ELSE
    // No latched run / inhibited / fault: ensure safe idle
    startSequenceRunning := FALSE;

    IF step <> 50 THEN
        lineContactor := FALSE;
    END_IF

    softstarterStart     := FALSE;
    softstarterContactor := FALSE;

    tonStartDelay(IN:=FALSE);
    tonOverlapDelay(IN:=FALSE);
    tonCurrentProof(IN:=FALSE);
    tonSSFbTimeout(IN:=FALSE);
    tonLineFbTimeout(IN:=FALSE);
    instTONSoftstartDelay(IN:=FALSE);

    IF NOT runLatch THEN
        deviceState := 'Idle (Parado)';
        step := 0;
    END_IF
END_IF


//────────────────────────────────────
// Blink generator (1 s ON / 1 s OFF)
// Gerador de pisca (1 s ligado / 1 s desligado)
//────────────────────────────────────
blinkTon(IN := TRUE, PT := T#1S);
IF blinkTon.Q THEN
    blinkTon(IN := FALSE);       // reset timer next cycle / reseta o timer no próximo ciclo
    blinkBit := NOT blinkBit;    // toggle blink bit / alterna o bit de pisca
END_IF


// =============================== Status code =======================================
// 0 = OFF
// 0-1 (alternando) = STARTING
// 1 = RUNNING
// 2 = FAULT
//==============================================================================
IF faultActive THEN
    // Fault has highest priority / Falha tem maior prioridade
    statusCode := 2;                             // FAULT

ELSIF softstarterContactor OR (softstarterContactor AND lineContactor)  THEN
    // STARTING: use blink (0/1) / PARTIDA: usa pisca (0/1)
    IF blinkBit THEN
        statusCode := 1;                         // ON (blink ON)
    ELSE
        statusCode := 0;                         // OFF (blink OFF)
    END_IF

ELSIF  lineContactor AND NOT softstarterContactor THEN
    // RUNNING: steady ON / EM FUNCIONAMENTO: ligado fixo
    statusCode := 1;                             // RUNNING

ELSE
    // OFF (stopped / idle) / Desligado (parado)
    statusCode := 0;                             // OFF
END_IF

END_FUNCTION_BLOCK

// ---- Function Blocks/PaperMachine/Auxiliary/FB_PressureControl_V1.TcPOU
(*
    FB_PressureControl_V1
    - Start pulse toggles run; Stop pulse/level forces stop
    - statusCode : INT (0=Idle, 1=Running, 2=Fault)
    - PID (OSCAT CTRL_PID) with optional reverse action
    - Input PT1 filter (OSCAT FT_PT1)
    - Engineering↔% scaling helper
    - VFD run supervision + analog feedback display (current, rpm)
    - Optional low/high pressure HOLD with hysteresis (normal-stop class)
*)

FUNCTION_BLOCK FB_PressureControl_V1
VAR_INPUT
    // ===== Sequence commands =====
    startCommand            : BOOL;            // Start pulse (toggle run)
    stopCommand             : BOOL;            // Stop pulse/level (force stop)

    // ===== Mode =====
    autoMode                : BOOL;            // TRUE=Automatic / FALSE=Manual
    reverseActing           : BOOL := FALSE;   // TRUE: increasing output decreases pressure (válvula); FALSE: direct (bomba)

    // ===== Process signals (PRESSURE) =====
    pressureFeedbackEng     : REAL;            // PV (engineering units) - Ex.: bar/kPa
    pressureSetpointEng     : REAL;            // SP (engineering units)

    // ===== Manual output (direct % to final element) =====
    manualOutputPct         : REAL;            // 0..100% manual output

    // ===== PID parameters (OSCAT CTRL_PID) =====
    kp                      : REAL := 1.0;     // proportional gain (magnitude; sign handled by reverseActing)
    tn                      : REAL := 8.0;     // integral time [s]
    tv                      : REAL := 0.0;     // derivative time [s]

    // ===== Output limits & offset =====
    outLowLimitPct          : REAL := 0.0;
    outHighLimitPct         : REAL := 100.0;
    outputOffsetPct         : REAL := 0.0;     // added to final output

    // ===== PID housekeeping =====
    resetPID                : BOOL;            // reset integrator

    // ===== Input filter (OSCAT PT1) =====
    enableInputFilter       : BOOL := TRUE;
    inputFilterTime         : TIME := T#300ms;
    inputFilterGainK        : REAL := 1.0;

    displayFilterTime       : TIME := T#20MS;	
	

    // ===== Optional scaling (engineering <-> %) =====
    enableScaling           : BOOL := TRUE;
    pLoEng                  : REAL := 0.0;     // e.g., 0 bar
    pHiEng                  : REAL := 10.0;    // e.g., 10 bar

    // ===== VFD interface & supervision =====
    vfdReady                : BOOL;            // VFD ready/healthy
    vfdRunFeedback          : BOOL;            // VFD RUN feedback
    vfdFaultFeedback        : BOOL;            // VFD fault feedback
    vfdRunFbTimeout         : TIME := T#5s;    // Timeout to receive RUN FB after start

    // ===== VFD analog feedbacks =====
    vfdCurrentFeedback      : REAL;            // Motor current [A]
    vfdEngFeedback          : REAL;            // Motor enginering feedback
    vfdTorqueFeedback       : REAL;            // Motor torque feedback
	

    // ===== SAFETY (true safety only) =====
    safetyOk                : BOOL := TRUE;    // Safety relay / chain OK
    estopOk                 : BOOL := TRUE;    // E-Stop loop OK
    guardClosedOk           : BOOL := TRUE;    // Doors/guards closed

    // ===== INTERLOCKS (process permissives) — NORMAL STOP ONLY =====
    interlock1              : BOOL := TRUE;
    interlock2              : BOOL := TRUE;
    interlock3              : BOOL := TRUE;
    interlock4              : BOOL := TRUE;
    interlock5              : BOOL := TRUE;
    interlock6              : BOOL := TRUE;

    // ===== Optional low-pressure supervision (normal-stop/hold) =====
    minPressureEnable       : BOOL := FALSE;   // Enable low-P hold
    minPressureStopEng      : REAL := 0.5;     // Trip threshold (Eng units) => stop & hold
    minPressureRestartEng   : REAL := 0.7;     // Release threshold (Eng units) => auto restart
    minPressureTripTime     : TIME := T#1s;    // P < Stop for this long to trip
    minPressureReleaseTime  : TIME := T#1s;    // P > Restart for this long to release

    // ===== Optional high-pressure supervision (normal-stop/hold) =====
    maxPressureEnable       : BOOL := FALSE;   // Enable high-P hold
    maxPressureStopEng      : REAL := 9.5;     // Trip threshold (Eng units)
    maxPressureRestartEng   : REAL := 9.2;     // Release threshold (Eng units)
    maxPressureTripTime     : TIME := T#1s;
    maxPressureReleaseTime  : TIME := T#1s;
END_VAR

VAR_OUTPUT
    running                 : BOOL;            // TRUE only in RUN (use to release other devices)
    controlOutputPct        : REAL;            // 0..100 %
    pidDiff                 : REAL;            // SET - ACT (post-scaling)
    pidLimited              : BOOL;            // TRUE if saturated
    deviceState             : STRING(80);      // Human-readable state (EN/PT-BR)
    vfdStartCmdOut          : BOOL;            // Asserted in Starting/Running (VFD START)

    // ===== Holds (normal stop class) =====
    minPressureHoldActive   : BOOL;
    maxPressureHoldActive   : BOOL;

    // Status & displays
    statusCode              : INT;             // 0=Idle, 1=Running, 2=Fault
    vfdCurrentDisplay       : REAL;            // Displayed motor current [A]
    vfdTorqueDisplay       : REAL;            // Displayed motor current [A]
    vfdEngDisplay           : REAL;            // Displayed motor speed [rpm]
	
END_VAR
VAR
    // ===== State & edges =====
    step                    : INT;             // 0=Idle,10=Starting,20=Running,90=Stopping
    startOld                : BOOL;
    stopOld                 : BOOL;
    rStart                  : BOOL;            // start pulse edge
    rStop                   : BOOL;            // stop pulse edge
    runLatch                : BOOL;            // toggled by Start; cleared by Stop

    // ===== Internals =====
    manualCmd               : REAL;
    yPID                    : REAL;
    kpUse                   : REAL;            // sign-adjusted Kp

    // Filtered PV (engineering)
    pressureFeedbackEngFilt : REAL;

    // PV/SP in %
    pvPct                   : REAL;
    spPct                   : REAL;

    // Timers / supervision
    tonRunFbWait            : TON;

    // Low/High pressure timers/flags
    tonMinPTrip             : TON;
    tonMinPRelease          : TON;
    tonMaxPTrip             : TON;
    tonMaxPRelease          : TON;

    // Instances
    instPID                 : CTRL_PID;
    instPT1                 : FT_PT1;

    // Aggregations
    allSafetyOK             : BOOL;
    anyInterlockOpen        : BOOL;
	
    instPT1_TorqueDisplay  		: FT_PT1;
    instPT1_SpeedDisplay   		: FT_PT1;
	
END_VAR

// ============================ Edges ============================
rStart := startCommand AND NOT startOld;
startOld := startCommand;

rStop  := stopCommand AND NOT stopOld;
stopOld := stopCommand;

// Start toggles run; Stop forces stop
IF rStart THEN
    runLatch := NOT runLatch;
END_IF;
IF rStop OR stopCommand THEN
    runLatch := FALSE;
END_IF;


// ============================ Aggregations =====================
allSafetyOK := safetyOk AND estopOk AND guardClosedOk;
anyInterlockOpen := NOT (interlock1 AND interlock2 AND interlock3 AND interlock4 AND interlock5 AND interlock6);

// Defaults each cycle
vfdStartCmdOut := FALSE;



// ============================ Pressure HOLD supervision ============================
// LOW-P
IF minPressureEnable THEN
    tonMinPTrip(IN := (pressureFeedbackEng <  minPressureStopEng),     PT := minPressureTripTime);
    tonMinPRelease(IN := (pressureFeedbackEng > minPressureRestartEng), PT := minPressureReleaseTime);
    IF tonMinPTrip.Q THEN minPressureHoldActive := TRUE; END_IF;
    IF tonMinPRelease.Q THEN minPressureHoldActive := FALSE; END_IF;
ELSE
    tonMinPTrip(IN := FALSE);
    tonMinPRelease(IN := FALSE);
    minPressureHoldActive := FALSE;
END_IF;

// HIGH-P
IF maxPressureEnable THEN
    tonMaxPTrip(IN := (pressureFeedbackEng > maxPressureStopEng),       PT := maxPressureTripTime);
    tonMaxPRelease(IN := (pressureFeedbackEng < maxPressureRestartEng), PT := maxPressureReleaseTime);
    IF tonMaxPTrip.Q THEN maxPressureHoldActive := TRUE; END_IF;
    IF tonMaxPRelease.Q THEN maxPressureHoldActive := FALSE; END_IF;
ELSE
    tonMaxPTrip(IN := FALSE);
    tonMaxPRelease(IN := FALSE);
    maxPressureHoldActive := FALSE;
END_IF;


// ============================ Immediate stop / safety/fault =======
IF rStop OR stopCommand THEN
    controlOutputPct := 0.0;
    running := FALSE;
    deviceState := 'Stopping (Stop command) / Parando (comando Stop)';
    runLatch := FALSE;
    step := 90;
END_IF;

IF vfdFaultFeedback THEN
    deviceState := 'Fault from VFD / Falha do inversor';
    runLatch := FALSE;
    step := 90;
END_IF;

IF NOT allSafetyOK THEN
    deviceState := 'Stopping: Safety chain open / Parando: segurança aberta';
    runLatch := FALSE;
    step := 90;
END_IF;


// ============================ State machine =====================
CASE step OF
    // ------------------------------------------------------------
    0: // Idle
        running := FALSE;
        controlOutputPct := 0.0;
        deviceState := 'Idle / Parado';
        vfdStartCmdOut := FALSE;

        // Start request via runLatch (toggled by Start pulse)
        IF runLatch AND NOT stopCommand THEN
            // Safety must be OK; VFD must be ready; pressure holds must be clear
            IF NOT allSafetyOK THEN
                deviceState := 'Start blocked: Safety not OK / Partida bloqueada: segurança NOK';
                runLatch := FALSE;
                step := 0;
            ELSIF NOT vfdReady THEN
                deviceState := 'Start blocked: VFD not ready / Partida bloqueada: inversor NOK';
                runLatch := FALSE;
                step := 0;
            ELSIF (minPressureEnable AND minPressureHoldActive) OR (maxPressureEnable AND maxPressureHoldActive) THEN
                deviceState := 'Start blocked: Pressure hold active / Partida bloqueada: hold de pressão';
                runLatch := FALSE;
                step := 0;
            ELSE
                deviceState := 'Starting / Partindo';
                vfdStartCmdOut := TRUE;                   // send START to VFD
                tonRunFbWait(IN := TRUE, PT := vfdRunFbTimeout);
                step := 10;
            END_IF
        END_IF

    // ------------------------------------------------------------
    10: // Starting (await RUN feedback)
        running := FALSE;
        deviceState := 'Starting (await RUN fb) / Aguardando RUN';
        vfdStartCmdOut := TRUE;

        // Safety/fault during start => stop
        IF NOT allSafetyOK THEN
            tonRunFbWait(IN := FALSE);
            deviceState := 'Stopping: Safety chain open';
            vfdStartCmdOut := FALSE;
            runLatch := FALSE;
            step := 90;

        ELSIF vfdFaultFeedback THEN
            tonRunFbWait(IN := FALSE);
            deviceState := 'Fault from VFD';
            vfdStartCmdOut := FALSE;
            runLatch := FALSE;
            step := 90;

        // Interlocks are normal stop only
        ELSIF anyInterlockOpen THEN
            tonRunFbWait(IN := FALSE);
            deviceState := 'Stopping: Interlock open / Intertravamento aberto';
            vfdStartCmdOut := FALSE;
            runLatch := FALSE;
            step := 90;

        // Pressure holds => normal stop
        ELSIF (minPressureEnable AND minPressureHoldActive) OR (maxPressureEnable AND maxPressureHoldActive) THEN
            tonRunFbWait(IN := FALSE);
            deviceState := 'Stopping: Pressure hold / Hold de pressão';
            vfdStartCmdOut := FALSE;
            runLatch := FALSE;
            step := 90;

        // RUN fb arrived
        ELSIF vfdRunFeedback THEN
            tonRunFbWait(IN := FALSE);
            step := 20;

        // Timeout
        ELSIF tonRunFbWait.Q THEN
            tonRunFbWait(IN := FALSE);
            deviceState := 'Start failed: RUN fb timeout / Tempo excedido RUN';
            vfdStartCmdOut := FALSE;
            runLatch := FALSE;
            step := 90;
        END_IF

    // ------------------------------------------------------------
    20: // Running (control loop)
        running := TRUE;               // release other devices with this
        deviceState := 'Running / Operando';
        vfdStartCmdOut := TRUE;

        // Supervision
        IF NOT allSafetyOK THEN
            deviceState := 'Stopping: Safety chain open';
            vfdStartCmdOut := FALSE;
            runLatch := FALSE;
            step := 90;

        ELSIF vfdFaultFeedback THEN
            deviceState := 'Fault from VFD';
            vfdStartCmdOut := FALSE;
            runLatch := FALSE;
            step := 90;

        ELSIF NOT vfdReady THEN
            deviceState := 'Stopping: VFD not ready';
            vfdStartCmdOut := FALSE;
            runLatch := FALSE;
            step := 90;

        ELSIF NOT vfdRunFeedback THEN
            deviceState := 'Stopping: RUN feedback lost';
            vfdStartCmdOut := FALSE;
            runLatch := FALSE;
            step := 90;

        // INTERLOCKS → NORMAL STOP ONLY
        ELSIF anyInterlockOpen THEN
            deviceState := 'Stopping: Interlock open';
            vfdStartCmdOut := FALSE;
            runLatch := FALSE;
            step := 90;

        // Pressure holds → NORMAL STOP
        ELSIF (minPressureEnable AND minPressureHoldActive) OR (maxPressureEnable AND maxPressureHoldActive) THEN
            deviceState := 'Stopping: Pressure hold';
            vfdStartCmdOut := FALSE;
            runLatch := FALSE;
            step := 90;

        // Start toggled OFF while running => stop
        ELSIF NOT runLatch THEN
            deviceState := 'Stopping (Start toggled off)';
            vfdStartCmdOut := FALSE;
            step := 90;

        ELSE
            // ---- Input filtering (PT1) ----
            IF enableInputFilter THEN
                instPT1(in := pressureFeedbackEng, T := inputFilterTime, K := inputFilterGainK, out => pressureFeedbackEngFilt);
            ELSE
                pressureFeedbackEngFilt := pressureFeedbackEng;
            END_IF

            // ---- Engineering -> % scaling ----
            IF enableScaling THEN
                pvPct := _ScaleToPct(pressureFeedbackEngFilt, pLoEng, pHiEng);
                spPct := _ScaleToPct(pressureSetpointEng,    pLoEng, pHiEng);
            ELSE
                pvPct := pressureFeedbackEngFilt;   // already %
                spPct := pressureSetpointEng;       // already %
            END_IF

            // ---- Manual path and PID with bumpless transfer ----
            manualCmd := LIMIT(0.0, manualOutputPct, 100.0);

            // Reverse/direct action by Kp sign
            IF reverseActing THEN
                kpUse := -ABS(kp);
            ELSE
                kpUse :=  ABS(kp);
            END_IF

            instPID(
                ACT := pvPct,
                SET := spPct,
                M_I := manualCmd,
                MAN := NOT autoMode,
                RST := resetPID,
                KP  := kpUse,
                TN  := tn,
                TV  := tv,
                LL  := outLowLimitPct,
                LH  := outHighLimitPct,
                Y   => yPID,
                DIFF=> pidDiff,
                LIM => pidLimited
            );

            // Mode select, offset, clamp
            IF autoMode THEN
                controlOutputPct := yPID;
            ELSE
                controlOutputPct := manualCmd;
            END_IF
            controlOutputPct := LIMIT(outLowLimitPct, controlOutputPct + outputOffsetPct, outHighLimitPct);
        END_IF

    // ------------------------------------------------------------
    90: // Stopping (normal, de-energize)
        running := FALSE;
        controlOutputPct := 0.0;
        vfdStartCmdOut := FALSE;
        tonRunFbWait(IN := FALSE);

        // Return to Idle once stop released and safety OK
        IF NOT stopCommand AND allSafetyOK THEN
            deviceState := 'Idle / Parado';
            step := 0;
        END_IF

    // ------------------------------------------------------------
    ELSE
        running := FALSE;
        controlOutputPct := 0.0;
        deviceState := 'Idle / Parado';
        vfdStartCmdOut := FALSE;
        step := 0;
END_CASE


// =============================== Status code =======================================
IF vfdFaultFeedback THEN
    statusCode := 2;             // Fault
ELSIF running THEN
    statusCode := 1;             // Running
ELSE
    statusCode := 0;             // Idle
END_IF

_FeedbackDisplay();

METHOD _FeedbackDisplay
VAR_INPUT
END_VAR
// 5) HMI DISPLAY SIGNALS (filtered speeds/torques + GROUP status)
instPT1_SpeedDisplay(in := vfdEngFeedback, T := displayFilterTime, K := 1.0, out => vfdEngDisplay);
instPT1_TorqueDisplay (in := vfdTorqueFeedback , T := displayFilterTime, K := 1.0, out => vfdTorqueDisplay);
END_METHOD

// ============================ Helper ============================
METHOD PRIVATE _ScaleToPct : REAL
VAR_INPUT
    xEng  : REAL;  // value in engineering units
    loEng : REAL;  // min eng
    hiEng : REAL;  // max eng
END_VAR
VAR
    span : REAL;
    pct  : REAL;
END_VAR

span := hiEng - loEng;
IF span = 0.0 THEN
    _ScaleToPct := 0.0; // avoid div by zero
ELSE
    pct := (xEng - loEng) / span * 100.0;
    _ScaleToPct := LIMIT(0.0, pct, 100.0);
END_IF
END_METHOD

END_FUNCTION_BLOCK

// ---- Function Blocks/PaperMachine/DriveControl/FB_FormingBoardControl_V1.TcPOU
FUNCTION_BLOCK FB_FormingBoardControl_V1
VAR_INPUT
    // ── Group / Interlocks ───────────────────────────────────────────────────────
    startGroup                   : BOOL;   // Start command (pulse / rising edge)
    stopGroup                    : BOOL;   // Stop command  (pressed / level)
    groupReset                   : BOOL;   // Group fault Reset (Comando reset falhas do grupo)
    groupFastStop           : BOOL;  // EN: Reset group faults / PT: Reset de falhas do grupo

    // ── VFD per-drive status inputs ─────────────────────────────────────────────
    formingBoardTractionRollFault               : BOOL;   // VFD ready/healthy (master)
	formingBoardTractionRollCoolingFault  : BOOL;   // VFD ready/healthy (master)
    formingBoardTractionRollVfdRunFeedback         : BOOL;   // VFD RUN feedback  (master)
    formingBoardTractionRollVfdFaultFeedback       : BOOL;   // VFD fault         (master)
   
	formingBoardSuctionRollFault                : BOOL;   // VFD ready/healthy (slave)
	formingBoardSuctionRollCoolingFault		: BOOL;   // VFD ready/healthy (slave)	
	
    formingBoardSuctionVfdRunFeedback          : BOOL;   // VFD RUN feedback  (slave)
    formingBoardSuctionVfdFaultFeedback        : BOOL;   // VFD fault         (slave)

	
	paperPresenceSensor				: BOOL;
	
    // ── Speed Setpoints ─────────────────────────────────────────────────────────
    groupAutoSpeedMPM            : REAL;   // Auto speed setpoint [m/min]
    groupMaxSpeed                : REAL := 600.0; // Max allowed line speed [m/min]

    // ── Auto / Manual ───────────────────────────────────────────────────────────
    groupSpeedAutoMan            : BOOL;   // 0=Manual / 1=Auto
    groupManualSpeedMPM          : REAL := 50.0;  // Manual speed [m/min]

    // ── Feedbacks ───────────────────────────────────────────────────────────────
    masterTorqueFeedback         : REAL;   // [% or Nm]
    slaveTorqueFeedback          : REAL;   // [% or Nm]
    masterSpeedFeedback          : REAL;   // [m/min or %] — be consistent
    slaveSpeedFeedback           : REAL;   // [m/min or %] — be consistent

    // ── Ratio & Offsets ─────────────────────────────────────────────────────────
    masterSlaveGearRatio		: REAL := 1.0;   // Slave/Master speed ratio
// 	interGroupGearRatio			: REAL := 1.0;   // Speed diference btween groups
	
    slaveTorqueOfsset            : REAL := 0.0;   // (typo kept) torque trim [%/Nm]
    slaveSpeedOffset             : REAL := 10;    // Offset as % of master speed (+5 => +5%)

    // ── Torque control parameters ───────────────────────────────────────────────
    torqueLimitMinPct            : REAL := 5.0;   // Min torque [%]  (allow negative if regen)
    torqueLimitMaxPct            : REAL := 100.0; // Max torque [%]
    torqueDeadbandPct            : REAL := 1.0;   // |torque| below => 0 (noise cleanup)
	
    torqueFilterTime             : TIME := T#1MS;
    displayFilterTime             : TIME := T#20MS;	

    // ── Dynamics (for ramp block) ───────────────────────────────────────────────
    rampRate                     : REAL := 0.01;  // Ref accel mag in %/s (A_UP=+rampRate, A_DN=-rampRate)

    // ── Speed difference limit ──────────────────────────────────────────────────
    speedDiferenceLimit          : REAL := 5.0;
	
	
	
	
	//Headbox inputs
	
	//==============================================================
	// FORMING BOARD — WIRE EDGE OVERRUN SENSORS
	//==============================================================
	formingBoardWireOverrunOperatorSideSensor : BOOL;  // TRUE when wire overruns on operator side
	formingBoardWireOverrunDriveSideSensor    : BOOL;  // TRUE when wire overruns on drive/motor side	

	//==============================================================
	// HEADBOX LIPS OPENING CONTROL — VARIABLES
	//==============================================================
	
	// Position feedback and physical limits [mm]
	headboxLipsPositionFeedback_mm     : REAL;          // Actual lips opening [mm]
	headboxLipsMinOpening_mm           : REAL := 0.0;   // Minimum allowed opening [mm]
	headboxLipsMaxOpening_mm           : REAL := 25.0;  // Maximum allowed opening [mm]
	
	// Limit sensors (digital inputs)
	headboxLipsLimitFullyOpen          : BOOL;          // TRUE when fully open (max) limit sensor active
	headboxLipsLimitFullyClosed        : BOOL;          // TRUE when fully closed (min) limit sensor active
	
	// Manual jog commands (for manual mode)
	headboxLipsManualOpenCmd           : BOOL;          // Jog open while pressed
	headboxLipsManualCloseCmd          : BOOL;          // Jog close while pressed
	
	// Automatic positioning (for auto mode)
	headboxLipsTargetSetpoint_mm       : REAL;          // Desired lips opening [mm]
	headboxLipsAutoAdjustCmd           : BOOL;          // Pulse to start auto adjustment
	
		
	formingBoardRollUpCmd        : BOOL;  // Command to move forming board UP (active-high)
	formingBoardRollDownCmd      : BOOL;  // Command to move forming board DOWN (active-high)
	formingBoardRollLimitUpSensor    : BOOL;  // TRUE when upper limit is reached (prevents further UP)
	formingBoardRollLimitDownSensor  : BOOL;  // TRUE when lower limit is reached (prevents further DOWN)
	formingBoardRollUpDownMotorFault            : BOOL;  // TRUE = fault present → disables all movement	
	
	formingBoardStretchCmd           : BOOL;  // Jog command to stretch (increase tension)
	formingBoardUnstretchCmd         : BOOL;  // Jog command to unstretch (decrease tension)
	formingBoardLimitStretchSensor   : BOOL;  // TRUE when maximum stretch limit is reached
	formingBoardLimitUnstretchSensor : BOOL;  // TRUE when minimum stretch limit is reached
	formingBoardStretchMotorFault         : BOOL;  // Fault interlock for stretch unit
	
		
END_VAR

VAR_OUTPUT
    deviceState                  : STRING;
    groupFault                   : BOOL;   // Fault present (Falha do grupo)

    // ── Drive References (0..100%) ──────────────────────────────────────────────
    masterDriveSpeedRefPct       : REAL;   // Master reference [%]
    slaveDriveSpeedRefPct        : REAL;   // Slave  reference [%]
	nextGroupSpeedRefPct		 : REAL;   // Next group reference [%]
	nextGroupSpeedRefMPM		 : REAL;   // Next group reference [Meters per minute]
	
    // ── Torque limit to slave (from master torque path / or PID) ───────────────
    slaveDriveTorqueLimit        : REAL;   // [% or Nm]

    // ── Drive Commands ──────────────────────────────────────────────────────────
    masterDriveEnable            : BOOL;
    slaveDriveEnable             : BOOL;
    masterDriveReset             : BOOL;
    slaveDriveReset              : BOOL;

    // ── Diagnostics ─────────────────────────────────────────────────────────────
    currentSpeedDifence          : REAL;

    // ── Group status & HMI displays ────────────────────────────────────────────
    statusCode                   	: INT;    // 0=Idle, 1=Starting, 2=Running, 3=Fault (group)
	
    masterSpeedMPMFilteredDisplay   : REAL;   // Filtered master speed [m/min]
    slaveSpeedMPMFilteredDisplay    : REAL;   // Filtered slave  speed [m/min]
	
    masterTorqueFilteredDisplay  	: REAL;   // Master torque (raw)  [% or Nm]
    slaveTorqueFilteredDisplay   	: REAL;   // Slave torque (filtered) [% or Nm]

    // ── NEW: per-drive motor status codes ───────────────────────────────────────
    masterStatusCode             : INT;    // 0=Idle, 1=Starting, 2=Running, 3=Fault
    slaveStatusCode              : INT;    // 0=Idle, 1=Starting, 2=Running, 3=Fault
	
	//==============================================================
	// HEADBOX LIPS OPENING CONTROL — OUTPUTS
	//==============================================================
	
	// Drive outputs (modulated by PWM in automatic mode)
	headboxLipsOpenCmd                : BOOL;  // Output to open lips (PWM-modulated in Auto mode)
	headboxLipsCloseCmd               : BOOL;  // Output to close lips (PWM-modulated in Auto mode)
	headboxLipsPosition_mm       		  : REAL;  // Target − Feedback error [mm]
	
	//==============================================================
	// FORMING BOARD — ROLL DRIVE OUTPUTS
	//==============================================================
	formingBoardRollUp       : BOOL;  // Output to drive the forming board UP
	formingBoardRollDown     : BOOL;  // Output to drive the forming board DOWN
	
	//==============================================================
	// FORMING BOARD — STRETCH DRIVE OUTPUTS
	//==============================================================
	formingBoardStretch      : BOOL;  // Output to stretch (increase tension)
	formingBoardUnstretch    : BOOL;  // Output to unstretch (decrease tension)
		

	hmiAlarms 				: PaperMachine_TypeHmiAlarms; 	

END_VAR

VAR
    // ── Internals / Ramps ───────────────────────────────────────────────────────
    rampTargetPct                : REAL;   // 0..100% target into ramp
    instFB_Gen_SRamp             : FB_Gen_SRamp; // Your ramp FB

    // ── State & Edges ───────────────────────────────────────────────────────────
    state                        : INT;    // 0=IDLE,1=ENABLE,2=WAIT_EN,3=RAMP_EN,4=RUN,5=STOPPING,10=FAULT
    startGroupOld                : BOOL;
    stopGroupOld                 : BOOL;
    rStart                       : BOOL;
    rStop                        : BOOL;

    // ── Timers & thresholds ─────────────────────────────────────────────────────
    instTONEnableWait            : TON;
    instTONStopWait              : TON;
    enableTimeout                : TIME := T#5s;  // Wait for op-enable
    stopTimeout                  : TIME := T#8s;  // Max wait to speed≈0
    speedZeroThresholdPct        : REAL := 4.00;  // Consider stopped if |speed| ≤ this
    epsRefPct                    : REAL := 0.05;  // Small epsilon for ref≈0

    // ── Ramp control ────────────────────────────────────────────────────────────
    rampReset                    : BOOL;   // Resets ramp (sets Y/V to 0 in your FB)

    // ── Filter state used by _TorqueReference ───────────────────────────────────
    torqueFiltY                  : REAL;   // last filtered torque
    torqueFiltInit               : BOOL;   // init flag (bumpless start)
    instsFT_PT1TorqueFilter      : FT_PT1;

    // ── Speed difference supervision ────────────────────────────────────────────
    instTONSpeedDifDelay         : TON;

    // ── HMI-only PT1 filters ───────────────────────────────────────────────────
    instPT1_MasterSpeedDisplay          : FT_PT1;
    instPT1_SlaveSpeedDisplay           : FT_PT1;
	
    instPT1_MasterTorqueDisplay  		: FT_PT1;
    instPT1_SlaveTorqueDisplay   		: FT_PT1;
	
	instFB_HeadboxLipsPWMControl		: FB_HeadboxLipsPWMControl;	
	
END_VAR

// ─────────────────────────────────────────────────────────────────────────────
// MAIN CALL SEQUENCE
// ─────────────────────────────────────────────────────────────────────────────
_FeedbackDisplay();
_GroupControl();          // 1) State machine: edges, enables, stop modes
_ReferenceGenerator();    // 2) Build master/slave references with ramp
_TorqueReference();       // 3) Legacy torque transfer (kept)
_StateDisplay();

_SpeedDifferenceCheck();  // 4) Speed difference monitor & trip
_headboxLipsPosition();

_auxiliaryControls();
_alarmsDisplay();

METHOD _alarmsDisplay
VAR_INPUT
END_VAR
//==============================================================
// FAULT EVALUATION — PER CONDITION (flags only; no global set)
//==============================================================

//----------------------------
// FORMING BOARD DRIVES
//----------------------------
hmiAlarms.formingBoardRollDriveFaultAlarm    := formingBoardRollUpDownMotorFault;
hmiAlarms.formingBoardStretchDriveFaultAlarm := formingBoardStretchMotorFault;

//----------------------------
// FORMING BOARD AUXILIARY MOTORS
//----------------------------
hmiAlarms.formingBoardSuctionRollFaultAlarm         := formingBoardSuctionRollFault;
hmiAlarms.formingBoardSuctionRollCoolingFaultAlarm  := formingBoardSuctionRollCoolingFault;
hmiAlarms.formingBoardTractionRollFaultAlarm        := formingBoardTractionRollFault;
hmiAlarms.formingBoardTractionRollCoolingFaultAlarm := formingBoardTractionRollCoolingFault;

//----------------------------
// FORMING BOARD WIRE OVERRUN
//----------------------------
hmiAlarms.formingBoardWireOverrunOperatorSideAlarm := formingBoardWireOverrunOperatorSideSensor;
hmiAlarms.formingBoardWireOverrunDriveSideAlarm    := formingBoardWireOverrunDriveSideSensor;

//----------------------------
// FORMING BOARD GROUP FAULT STATUS
//----------------------------
groupFault :=
    hmiAlarms.formingBoardRollDriveFaultAlarm OR
    hmiAlarms.formingBoardStretchDriveFaultAlarm OR
    hmiAlarms.formingBoardSuctionRollFaultAlarm OR
    hmiAlarms.formingBoardSuctionRollCoolingFaultAlarm OR
    hmiAlarms.formingBoardTractionRollFaultAlarm OR
    hmiAlarms.formingBoardTractionRollCoolingFaultAlarm OR
    hmiAlarms.formingBoardWireOverrunOperatorSideAlarm OR
    hmiAlarms.formingBoardWireOverrunDriveSideAlarm;
END_METHOD

METHOD _auxiliaryControls
VAR_INPUT
END_VAR
//============================
// FORMING BOARD ROLL UP/DOWN
//============================
IF NOT formingBoardRollUpDownMotorFault THEN
    IF formingBoardRollUpCmd AND NOT formingBoardRollDownCmd AND NOT formingBoardRollLimitUpSensor THEN
        formingBoardRollUp := TRUE;
    ELSE
        formingBoardRollUp := FALSE;
    END_IF;

    IF formingBoardRollDownCmd AND NOT formingBoardRollUpCmd AND NOT formingBoardRollLimitDownSensor THEN
        formingBoardRollDown := TRUE;
    ELSE
        formingBoardRollDown := FALSE;
    END_IF;
ELSE
    formingBoardRollUp := FALSE;
    formingBoardRollDown := FALSE;
END_IF;


//============================
// FORMING BOARD STRETCH/UNSTRETCH
//============================
IF NOT formingBoardStretchMotorFault THEN
    IF formingBoardStretchCmd AND NOT formingBoardUnstretchCmd AND NOT formingBoardLimitStretchSensor THEN
        formingBoardStretch := TRUE;
    ELSE
        formingBoardStretch := FALSE;
    END_IF;

    IF formingBoardUnstretchCmd AND NOT formingBoardStretchCmd AND NOT formingBoardLimitUnstretchSensor THEN
        formingBoardUnstretch := TRUE;
    ELSE
        formingBoardUnstretch := FALSE;
    END_IF;
ELSE
    formingBoardStretch := FALSE;
    formingBoardUnstretch := FALSE;
END_IF;
END_METHOD

METHOD _FeedbackDisplay
VAR_INPUT
END_VAR
// 5) HMI DISPLAY SIGNALS (filtered speeds/torques + GROUP status)
instPT1_MasterSpeedDisplay(in := masterSpeedFeedback, T := displayFilterTime, K := 1.0, out => masterSpeedMPMFilteredDisplay);
instPT1_SlaveSpeedDisplay (in := slaveSpeedFeedback , T := displayFilterTime, K := 1.0, out => slaveSpeedMPMFilteredDisplay);

instPT1_MasterTorqueDisplay(in := masterTorqueFeedback, T := displayFilterTime, K := 1.0, out => masterTorqueFilteredDisplay);
instPT1_SlaveTorqueDisplay (in := slaveTorqueFeedback , T := displayFilterTime, K := 1.0, out => slaveTorqueFilteredDisplay);
END_METHOD

// ============================== Methods ==============================
// 1) GROUP CONTROL
METHOD _GroupControl
VAR_INPUT
END_VAR
VAR
    speedsNearZero : BOOL;
    refNearZero    : BOOL;
    bothOpEnabled  : BOOL;
END_VAR
// Edges
rStart := startGroup AND NOT startGroupOld;     // Start on pulse
rStop  := stopGroup  AND NOT stopGroupOld;      // Stop also has an edge
startGroupOld := startGroup;
stopGroupOld  := stopGroup;

// Feedback conditions (unit matches your % references)
speedsNearZero :=
    (ABS(masterSpeedFeedback) <= speedZeroThresholdPct) AND
    (ABS(slaveSpeedFeedback)  <= speedZeroThresholdPct);

// Also consider the reference near zero (backup)
refNearZero := ABS(masterDriveSpeedRefPct) <= epsRefPct;

// Use the original "operation enabled" for RUN readiness
bothOpEnabled := formingBoardTractionRollFault AND formingBoardSuctionRollFault;

CASE state OF
    0: // IDLE
        deviceState := 'IDLE';
        rampReset := TRUE;
        IF rStart AND NOT groupFault THEN
            state := 1;
        END_IF

    1: // ENABLE DRIVES
        deviceState := 'ENABLE_DRIVES';
        masterDriveEnable := TRUE;
        slaveDriveEnable  := TRUE;
        rampReset         := TRUE;

        instTONEnableWait(IN := TRUE, PT := enableTimeout);
        IF stopGroup THEN
            instTONEnableWait(IN := FALSE);
            state := 5;
        ELSE
            state := 2;
        END_IF

    2: // WAIT ENABLE FEEDBACK
        deviceState := 'WAIT_ENABLE_FEEDBACK';
        masterDriveEnable := TRUE;
        slaveDriveEnable  := TRUE;
        rampReset         := TRUE;

        instTONEnableWait(IN := TRUE, PT := enableTimeout);

        IF groupFault THEN
            instTONEnableWait(IN := FALSE);
            state := 10;
        ELSIF rStop OR stopGroup THEN
            instTONEnableWait(IN := FALSE);
            state := 5;
        ELSIF bothOpEnabled THEN
            instTONEnableWait(IN := FALSE);
            state := 3;
        ELSIF instTONEnableWait.Q THEN
            instTONEnableWait(IN := FALSE);
            state := 10; // fault: no enable feedback
        END_IF

    3: // RAMP ENABLE (single-cycle gate)
        deviceState := 'RAMP_ENABLE';
        masterDriveEnable := TRUE;
        slaveDriveEnable  := TRUE;
        rampReset         := FALSE; // release ramp now
        IF stopGroup THEN
            state := 5;
        ELSE
            state := 4;
        END_IF

    4: // RUN
        deviceState := SEL(groupSpeedAutoMan,'RUN (Manual)', 'RUN (Auto)');
        masterDriveEnable := TRUE;
        slaveDriveEnable  := TRUE;
        rampReset         := FALSE;

        IF groupFault THEN
            state := 10;
        ELSIF rStop OR stopGroup THEN
            state := 5;
        END_IF

    5: // STOPPING (controlled)
        deviceState := 'STOPPING';
        masterDriveEnable := TRUE;    // keep enabled during decel
        slaveDriveEnable  := TRUE;
        rampReset         := FALSE;   // ramp down references
        // instTONStopWait(IN := TRUE, PT := stopTimeout);  // optional timeout

        // Disable when speed≈0 AND reference≈0
        IF groupFault THEN
            instTONStopWait(IN := FALSE);
            state := 10;

        ELSIF speedsNearZero AND refNearZero THEN
            masterDriveEnable := FALSE;
            slaveDriveEnable  := FALSE;
            instTONStopWait(IN := FALSE);
            state := 0;

        ELSIF instTONStopWait.Q THEN
            masterDriveEnable := FALSE;
            slaveDriveEnable  := FALSE;
            instTONStopWait(IN := FALSE);
            state := 10;
        END_IF

    10: // FAULT
        deviceState := 'FAULT';
        rampReset         := TRUE;    // force ramp outputs to zero
        masterDriveEnable := FALSE;
        slaveDriveEnable  := FALSE;

        // Clear fault when fault disappears and start is low
        IF (NOT groupFault) AND (NOT startGroup) THEN
            state := 0;
        END_IF
END_CASE;
END_METHOD

METHOD _headboxLipsPosition
VAR_INPUT
END_VAR
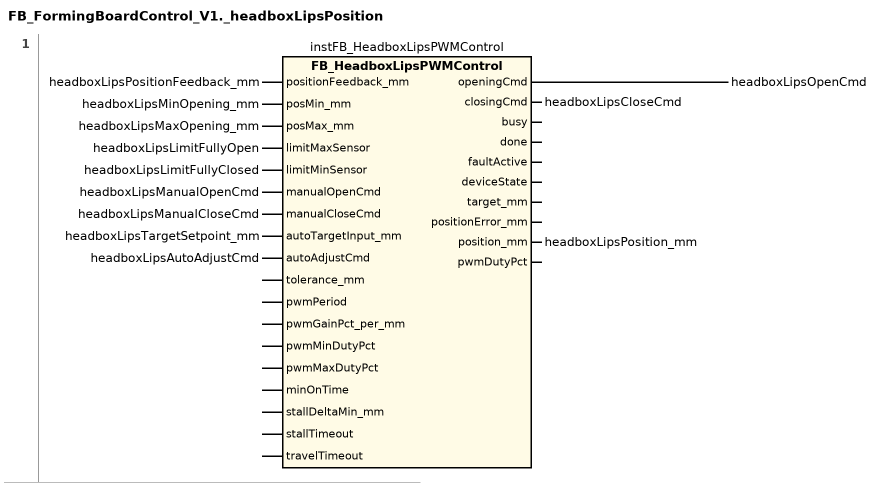
// NETWORK 1
instFB_HeadboxLipsPWMControl(
    positionFeedback_mm := headboxLipsPositionFeedback_mm,
    posMin_mm := headboxLipsMinOpening_mm,
    posMax_mm := headboxLipsMaxOpening_mm,
    limitMaxSensor := headboxLipsLimitFullyOpen,
    limitMinSensor := headboxLipsLimitFullyClosed,
    manualOpenCmd := headboxLipsManualOpenCmd,
    manualCloseCmd := headboxLipsManualCloseCmd,
    autoTargetInput_mm := headboxLipsTargetSetpoint_mm,
    autoAdjustCmd := headboxLipsAutoAdjustCmd,
    closingCmd => headboxLipsCloseCmd,
    position_mm => headboxLipsPosition_mm); // FB_HeadboxLipsPWMControl
headboxLipsOpenCmd := instFB_HeadboxLipsPWMControl.openingCmd;
END_METHOD

// 2) REFERENCE GENERATOR
METHOD _ReferenceGenerator
VAR
    headroomEpsPct      : REAL := 0.20;   // anti-chatter near 100%
    offsetPct           : REAL;
    denom               : REAL;
    maxMasterBySlave    : REAL;
    allowedCapPct       : REAL;
    currMasterPct       : REAL;
    currSlavePct        : REAL;
    targetPct           : REAL;
    cmdSpeedMPM         : REAL;
END_VAR
// 1) Select Auto/Manual command (MPM)
IF groupSpeedAutoMan THEN
    cmdSpeedMPM := groupAutoSpeedMPM;
ELSE
    cmdSpeedMPM := groupManualSpeedMPM;
END_IF

// 2) Scale to 0..100% for the drives
targetPct := _Scale(
    X    := cmdSpeedMPM,
    I_LO := 0.0,          I_HI := groupMaxSpeed,
    O_LO := 0.0,          O_HI := 100.0);

// 3) During STOPPING/FAULT we want zero target; in STOPPING we still ramp down
IF state = 5 THEN
    rampTargetPct := 0.0;
ELSE
    rampTargetPct := targetPct;
END_IF

// --- Pre-limit so SLAVE can’t exceed 100% for given gear + offset ---
offsetPct := slaveSpeedOffset * 0.01;
denom     := masterSlaveGearRatio + offsetPct;

// If denom <= 0, fall back to 100% (no additional cap required)
IF denom > 0.0 THEN
    maxMasterBySlave := 100.0 / denom;   // master % that makes slave hit 100%
ELSE
    maxMasterBySlave := 100.0;
END_IF;

// The cap the master target must obey (also respect master’s own 100%)
allowedCapPct := MIN(100.0, maxMasterBySlave);

// Apply cap to upward commands only (don’t block decel)
rampTargetPct := MIN(rampTargetPct, allowedCapPct);

// --- Freeze upward if currently at/near limit (anti-overrun using current refs) ---
currMasterPct := instFB_Gen_SRamp.Y;                          // current master ref (%)
currSlavePct  := LIMIT(0.0, currMasterPct * (masterSlaveGearRatio + offsetPct), 100.0);

IF (currMasterPct >= 100.0 - headroomEpsPct) OR
   (currSlavePct  >= 100.0 - headroomEpsPct) THEN
    // Prevent increasing the target above current value; allow decreases
    rampTargetPct := MIN(rampTargetPct, currMasterPct);
END_IF

// 4) Ramp call (unchanged)
instFB_Gen_SRamp(
    X          := rampTargetPct,
    A_UP       := MAX(0.0, rampRate),
    A_DN       := -MAX(0.0, rampRate),
    VU_MAX     := 1000.0,
    VD_MAX     := -1000.0,
    LIMIT_HIGH := 100.0,
    RST        := rampReset);

IF state = 5 THEN
    instFB_Gen_SRamp.LIMIT_LOW := 0.0;
ELSE
    instFB_Gen_SRamp.LIMIT_LOW := 3.5;
END_IF

// 5) Master reference = ramp Y but also respect the slave-driven cap
masterDriveSpeedRefPct := MIN(instFB_Gen_SRamp.Y, allowedCapPct);

// 6) Slave reference: gear + offset, then clamp 0..100
slaveDriveSpeedRefPct :=
    LIMIT(0.0, masterDriveSpeedRefPct * (masterSlaveGearRatio + offsetPct), 100.0);

// 7) Final safety clamp for master (symmetry) + forward as % to next group
masterDriveSpeedRefPct := LIMIT(0.0, masterDriveSpeedRefPct, 100.0);
nextGroupSpeedRefPct   := masterDriveSpeedRefPct;

// 8) Also forward the next group reference in MPM (easy to replicate elsewhere)
nextGroupSpeedRefMPM := _Scale(
    X    := nextGroupSpeedRefPct,
    I_LO := 0.0,          I_HI := 100.0,
    O_LO := 0.0,          O_HI := groupMaxSpeed);
END_METHOD

METHOD PRIVATE _Scale : REAL
VAR_INPUT
    X    : REAL;
    I_LO : REAL;
    I_HI : REAL;
    O_LO : REAL;
    O_HI : REAL;
END_VAR
IF I_LO = I_HI THEN
	_Scale := O_LO;
ELSE
	_Scale := (O_HI - O_LO) / (I_HI - I_LO) * (LIMIT(I_LO, X, I_HI) - I_LO) + O_LO;
END_IF;
END_METHOD

// 6) OPTIONAL: SLAVE TORQUE PID TRACKING (new)
METHOD _SlaveTorquePID
VAR_INPUT
    enablePID : BOOL := TRUE;   // TRUE=PID active, FALSE=hold/track current output
    Kp        : REAL := 0.8;    // proportional gain (tune as needed)
    Tn        : REAL := 1.5;    // integral time [s]
    Tv        : REAL := 0.0;    // derivative time [s]
END_VAR
VAR
    masterFilt : REAL;
    slaveFilt  : REAL;
    sp         : REAL;  // setpoint (master)
    pv         : REAL;  // process value (slave)
    y          : REAL;  // PID output (pre-clamp)
    e          : REAL;  // SET - ACT (diagnostic)
    limMin     : REAL;
    limMax     : REAL;
END_VAR
VAR_STAT
    pid        : CTRL_PID;  // PID instance (retained)
    fMaster    : FT_PT1;    // PT1 for master torque
    fSlave     : FT_PT1;    // PT1 for slave torque
END_VAR
// 1) Filter master & slave torques (reuse existing time constant)
fMaster(in := masterTorqueFeedback, T := torqueFilterTime, K := 1.0, out => masterFilt);
fSlave (in := slaveTorqueFeedback , T := torqueFilterTime, K := 1.0, out => slaveFilt);

// 2) Build setpoint and PV
sp := masterFilt + slaveTorqueOfsset;   // follow master + configured trim
pv := slaveFilt;

// 3) Limits from existing configuration
limMin := torqueLimitMinPct;
limMax := torqueLimitMaxPct;

// 4) PID with bumpless transfer (manual input tracks current output when disabled)
pid(
    ACT := pv,                      // process value (slave torque)
    SET := sp,                      // setpoint (master torque)
    MAN := NOT enablePID,           // MAN=TRUE => manual/track
    M_I := slaveDriveTorqueLimit,   // track current output for bumpless re-enable
    RST := FALSE,                   // external reset (unused)
    KP  := Kp,
    TN  := Tn,
    TV  := Tv,
    LL  := limMin,
    LH  := limMax,
    Y   => y,
    DIFF=> e,
    LIM =>                          // unused
);

// 5) Clamp and publish
slaveDriveTorqueLimit := LIMIT(limMin, y, limMax);
END_METHOD

METHOD PRIVATE _SpeedDifferenceCheck
VAR
    diff : REAL;
END_VAR
// 1) Absolute difference Master-Slave
diff := ABS(masterSpeedMPMFilteredDisplay - slaveSpeedMPMFilteredDisplay);
currentSpeedDifence := diff;

// 2) If beyond limit -> stop group (with a small delay)
IF diff > speedDiferenceLimit THEN
    instTONSpeedDifDelay.IN := TRUE;
    instTONSpeedDifDelay.PT := T#2S;

    IF instTONSpeedDifDelay.Q THEN
        state := 10;                  // Fault
        deviceState := 'FAULT: Speed difference exceeded';
    END_IF
ELSE
    instTONSpeedDifDelay.IN := FALSE;
END_IF

instTONSpeedDifDelay();
END_METHOD

METHOD _StateDisplay
VAR_INPUT
END_VAR

// ──────────────────────────────────────────────────────────────────────────────
// _StateDisplay
// Maps the internal machine "state" to a compact HMI status code and derives
// per-drive motor status codes from VFD signals.
//
// statusCode / masterStatusCode / slaveStatusCode legend:
//   0 = Idle, 1 = Starting, 2 = Running, 3 = Fault
//
// Machine "state" groups:
//   0 = IDLE, 1 = ENABLE, 2 = WAIT_EN, 3 = RAMP_EN, 4 = RUN, 5 = STOPPING, 10 = FAULT
// Priority rule (for motors): Fault > Running > Starting > Idle
// ──────────────────────────────────────────────────────────────────────────────
VAR CONSTANT
    STATUS_IDLE     : INT := 0;
//    STATUS_STARTING : INT := 1;
    STATUS_RUNNING  : INT := 1;
    STATUS_FAULT    : INT := 2;
END_VAR

// ─────────────── Group machine states into a single HMI statusCode ───────────
CASE state OF
    10: // FAULT
        statusCode := STATUS_FAULT;

    4:  // RUN
        statusCode := STATUS_RUNNING;

    1, 2, 3: // ENABLE / WAIT_EN / RAMP_EN
//        statusCode := STATUS_STARTING;

    ELSE // IDLE, STOPPING, or any other unlisted state
        statusCode := STATUS_IDLE;
END_CASE;

// ─────────────── Helper pattern for per-drive status (inline) ────────────────
// Evaluation order enforces priority: Fault > Running > Starting > Idle

// Master drive
IF formingBoardTractionRollVfdFaultFeedback THEN
    masterStatusCode := STATUS_FAULT;
ELSIF formingBoardTractionRollVfdRunFeedback THEN
    masterStatusCode := STATUS_RUNNING;
ELSE
    masterStatusCode := STATUS_IDLE;
END_IF;

// Slave drive
IF formingBoardSuctionVfdFaultFeedback THEN
    slaveStatusCode := STATUS_FAULT;
ELSIF formingBoardSuctionVfdRunFeedback THEN
    slaveStatusCode := STATUS_RUNNING;
ELSE
    slaveStatusCode := STATUS_IDLE;
END_IF;
END_METHOD

METHOD _TorqueReference
VAR
    rawTorque     : REAL;
    filtTorque    : REAL;
    torqueCmd     : REAL;
    limitedTorque : REAL;
    clamped       : BOOL;
END_VAR
// 1) Read master torque (keep units consistent with your limits)
rawTorque := masterTorqueFeedback;

// 2) Low-pass filter (OSCAT PT1)
instsFT_PT1TorqueFilter(
    in  := rawTorque,
    T   := torqueFilterTime,   // time constant in seconds (e.g., 0.25)
    K   := 0.8,                // unity gain
    out => filtTorque
);

// 3) Deadband cleanup
IF ABS(filtTorque) < torqueDeadbandPct THEN
    filtTorque := 0.0;
END_IF

// 4) Apply offset between master and slave
torqueCmd := filtTorque + slaveTorqueOfsset;

// 5) Clamp to limits
limitedTorque := LIMIT(torqueLimitMinPct, torqueCmd, torqueLimitMaxPct);
clamped       := (limitedTorque <> torqueCmd);

// 6) Output
slaveDriveTorqueLimit := limitedTorque;


//slaveDriveTorqueLimit := LIMIT(torqueLimitMinPct, masterTorqueFeedback, torqueLimitMaxPct);
END_METHOD

END_FUNCTION_BLOCK

// ---- Function Blocks/PaperMachine/Auxiliary/FB_MixPumpControl_V1.TcPOU
(*
===============================================================================
FB_MixPumpControl_V1  —  Rev.2025-09-07

CHANGE LOG
- Start/Stop harmonizado com FB_PressureControl_V1:
  • Detecção de borda (start/stop), latch de RUN, interlocks como parada normal,
    timeout para vfdRunFeedback, passos: Idle(0) → Starting(10) → Running(20) → Stopping(90) → Idle.
  • Parada imediata em falha/stop; parada normal por interlock/processo.
- Novas variáveis (HMI):
  • statusCode : INT  // 0=Idle, 1=Starting, 2=Running, 3=Fault
  • vfdCurrentDisplay : REAL  // corrente filtrada (A ou %)
  • vfdTorqueDisplay  : REAL  // torque filtrado (Nm ou %)
  • (mapear de vfdCurrentFeedback / vfdTorqueFeedback; se não conectados, exibem 0.0)
- Reorganização/limpeza (sem mudar função):
  • Execução do PID/auto-man, filtro PV e cálculo de setpoint automático
    executados no estado RUN; resets/segurança centralizados.
  • Comentários EN + (pt-BR) nas adições.

STATE DIAGRAM (textual)
Idle(0) --Start→ Starting(10) --RUN fb→ Running(20)
Running(20) --Stop/Interlock/Hold→ Stopping(90) → Idle(0)
Any state --Fault/Safety→ Stopping(90) → Idle(0)
Fault code mapping: statusCode=3 quando falha; Stopping mapeia para Idle (0) ao finalizar.

NOTAS DE MAPEAMENTO
- Displays:
  vfdCurrentDisplay <= vfdCurrentFeedback (PT1 curto)  // (corrente)
  vfdTorqueDisplay  <= vfdTorqueFeedback  (PT1 curto)  // (torque)
- Se os nomes reais dos sinais forem diferentes (ex.: iVfd, torqueVfdPct),
  conecte-os às novas entradas vfdCurrentFeedback / vfdTorqueFeedback conforme o seu projeto.
===============================================================================
*)

FUNCTION_BLOCK FB_MixPumpControl_V1
VAR_INPUT
    // ===== Commands =====
    startCommand               : BOOL;    // Start pulse (toggle run) (Pulso de partida alterna RUN)
    stopCommand                : BOOL;    // Stop pulse/level (Parada)
    autoMode                   : BOOL;    // TRUE=Auto / FALSE=Manual (Modo automático)

    // ===== Process feedbacks / tuning =====
    pressureFeedback_mmH2O     : REAL;    // PV [mmH2O]
	manualSetpointInc            : BOOL;    // Manual output 0..100% (Saída manual)
    manualSetpointDec            : BOOL;    // Manual output 0..100% (Saída manual)

    formingBoardSpeedMPM       : REAL;    // Wire speed [m/min] (Velocidade da tela)

    jetToWireRatioInc          : BOOL;    // Increment ratio (Incrementa razão)
    jetToWireRatioDec          : BOOL;    // Decrement ratio (Decrementa razão)
    jetToWireRatioMin          : REAL := 0.5;
    jetToWireRatioMax          : REAL := 2.0;
    jetToWireRatioStep         : REAL := 0.01;

    jetHeadGainK               : REAL := 1.0;    // Gain on computed head (Ganho no head calculado)
    jetHeadOffset_mmH2O        : REAL := 0.0;    // Offset [mmH2O] (Offset no head)
    minAutoSP_mmH2O            : REAL := 0.0;    // Clamp low [mmH2O] (Limite inferior)
    maxAutoSP_mmH2O            : REAL := 4000.0; // Clamp high [mmH2O] (Limite superior)

    // ===== PID params (OSCAT CTRL_PID) =====
    kp                         : REAL := 0.8;
    tn                         : REAL := 3.0;
    tv                         : REAL := 0.0;
    pidDeadband_mmH2O          : REAL := 5.0;    // SUP (faixa morta no DIFF em mmH2O)
    outLowLimitPct             : REAL := 0.0;    // LL
    outHighLimitPct            : REAL := 100.0;  // LH
    outputOffsetPct            : REAL := 0.0;    // OFS
    resetPID                   : BOOL;           // RST

    // ===== PV input filter =====
    enableInputFilter          : BOOL := TRUE;
    inputFilterTime            : TIME := T#300ms;
    inputFilterGainK           : REAL := 1.0;

    // ===== Interlocks (normal stop only) =====
    interlock1                 : BOOL;   // Interlock/permissive (Intertravamento)
    interlock2                 : BOOL;
    interlock3                 : BOOL;
    interlock4                 : BOOL;

    // ===== VFD feedbacks & supervision =====
    vfdReady                   : BOOL;   // VFD ready/healthy (Pronto)
    vfdRunFeedback             : BOOL;   // VFD RUN FB (Confirmação de RUN)
    vfdFaultFeedback           : BOOL;   // VFD Fault (Falha inversor)
    vfdRunFbTimeout            : TIME := T#5s;   // Timeout to receive RUN FB

    // ===== VFD analog feedbacks =====
    vfdCurrentFeedback      : REAL;            // Motor current [A]
    vfdEngFeedback          : REAL;            // Motor enginering feedback
    vfdTorqueFeedback       : REAL;            // Motor torque feedback

	
END_VAR

VAR_OUTPUT
    // ===== Machine state =====
    running                    : BOOL;            // TRUE in RUN (libera outros dispositivos)
    faultActive                : BOOL;            // Latched fault (Falha memorizada)
    deviceState                : STRING(80);      // Human-readable (EN/PT-BR)
    vfdStartCmd                : BOOL;            // RUN command (Comando de partida ao inversor)

    // ===== Drive reference / control =====
    vfdSpeedPct                : REAL;            // 0..100% speed reference

    // ===== Jet-to-wire & pressure calc =====
//    jetToWireRatio             : REAL;            // Current ratio
    jetSpeed_mps               : REAL;            // Computed jet speed [m/s]
    headBoxMMH2OCalc           : REAL;            // Auto SP to PID [mmH2O]
    headBoxMMH2ORead           : REAL;            // PV filtered (para HMI)

    // ===== PID observability =====
    pidDiff                    : REAL;            // DIFF (deadband-filtered)
    pidLimited                 : BOOL;            // TRUE se Y saturado

    // ===== (NEW) HMI displays =====
//    manualSetpoint            : REAL;    		// Manual output 0..100% (Saída manual)	
    statusCode                 : INT;             // 0=Idle,1=Starting,2=Running,3=Fault
    vfdCurrentDisplay          : REAL;            // corrente (A ou %), filtrada para HMI
    vfdTorqueDisplay           : REAL;            // torque (Nm ou %), filtrado para HMI
    vfdEngDisplay           	: REAL;            // Displayed motor speed [rpm]	
	
END_VAR

VAR
	
	// ====== Edges & state-latch (bordas e trava de RUN) ======
    firstScan : BOOL := TRUE;   // TRUE only on first PLC cycle (Primeira varredura)
	
    // ====== Edges & state-latch (bordas e trava de RUN) ======
    startOld                   : BOOL;
    stopOld                    : BOOL;
    rStart                     : BOOL;
    rStop                      : BOOL;
    runLatch                   : BOOL;     // toggled by Start, cleared by Stop/Fault (Trava de execução)

    // ====== Step machine ======
    step                       : INT;      // 0=Idle,10=Starting,20=Running,90=Stopping

    // ====== Helpers ======
    allInterlocksOK            : BOOL;
    yPID_Pct                   : REAL;
    manualCmdPct               : REAL;
    filteredPV_mmH2O           : REAL;
    faultMsg                   : STRING(80);

    // ====== Timers ======
    tonRunFbWait               : TON;      // Wait RUN FB after start (Aguardar RUN do VFD)

    // ====== Instances already used in original FB ======
    instPID                    : CTRL_PID; // OSCAT PID
    instsFT_PT1TInputFilter    : FT_PT1;   // PT1 para PV

    // ====== (NEW) Display PT1 filters (pequeno Tc) ======
    instPT1_CurrentDisplay     : FT_PT1;   // PT1 para corrente exibida
    instPT1_TorqueDisplay      : FT_PT1;   // PT1 para torque exibido
	instPT1_SpeedDisplay		: FT_PT1;   // PT1 para torque exibido
	
    displayFilterTime          : TIME := T#50ms; // Small smoothing (Suavização leve)
	jetToWireRatioOld: REAL;
	manualSetpointOld: REAL;
	instTON_RunningDelay: TON;
END_VAR

VAR PERSISTENT
    // Mantido do original (tuner de razão)
    instTUNE2RatioSetpoint     : TUNE2;   // Ratio tuner with min/max clamp
  	instTUNE2ManSetpoint     	: TUNE2;   // Ratio tuner with min/max clamp

END_VAR

VAR_IN_OUT
	
    jetToWireRatio             : REAL;            // Current ratio
    manualSetpoint            : REAL;    		// Manual output 0..100% (Saída manual)	
	

END_VAR

// ============================ INITIALIZATION ============================
// Run this block only once on first cycle (Executa apenas uma vez)
IF firstScan THEN

	jetToWireRatio := instTUNE2RatioSetpoint.Y;
	manualSetpoint := instTUNE2ManSetpoint.Y;
	jetToWireRatioOld := jetToWireRatio;
	manualSetpointOld := manualSetpoint;
    firstScan := FALSE;             // Clear after first execution
	
END_IF




// ============================== MAIN EXECUTION ==============================
(* --------- 1) Edge detection (detecção de borda) --------- *)
rStart := startCommand AND NOT startOld;
startOld := startCommand;

rStop  := stopCommand AND NOT stopOld;
stopOld := stopCommand;

// Start toggles run; Stop forces stop (Start alterna RUN; Stop força parada)
IF rStart THEN
    runLatch := TRUE;
END_IF;
IF rStop OR stopCommand THEN
    runLatch := FALSE;
END_IF;

// --------- 2) Aggregations / defaults ---------
allInterlocksOK := interlock1 AND interlock2 AND interlock3 AND interlock4;

// Defaults every cycle (padrões por ciclo)
vfdStartCmd   := FALSE;
deviceState   := 'Idle / Parado';

// --------- 3) Immediate stops/faults (paradas/falhas imediatas) ---------
IF vfdFaultFeedback THEN
    // Inversor sinalizou falha => parar imediatamente
    faultActive := TRUE;
    faultMsg := 'Fault: VFD fault feedback / Falha: inversor';
    runLatch := FALSE;
    step := 90;  // Stopping
END_IF;

IF rStop OR stopCommand THEN
    // Comando de parada (classe normal, mas imediato no comando)
    runLatch := FALSE;
    step := 90;  // Stopping
END_IF;

// --------- 4) State machine (máquina de estados) ---------
CASE step OF
    // ============================= 0) IDLE =============================
    0:
        running     := FALSE;
        vfdStartCmd := FALSE;
        vfdSpeedPct := 0.0;
        deviceState := 'Idle / Parado';

        // Limpar timeout e mensagens
        tonRunFbWait(IN := FALSE);
        IF NOT startCommand AND NOT stopCommand THEN
            // libera falha quando em repouso sem comandos
            faultActive := FALSE;
            faultMsg := '';
        END_IF

        // Pedido de partida via runLatch
        IF runLatch AND NOT stopCommand THEN
            IF NOT vfdReady THEN
                deviceState := 'Start blocked: VFD not ready / Partida bloqueada: inversor NOK';
                runLatch := FALSE; // rejeita pedido
            ELSIF NOT allInterlocksOK THEN
                deviceState := 'Start blocked: interlock open / Partida bloqueada: intertravamento';
                runLatch := FALSE;
            ELSE
                // Tudo OK => partir
                deviceState := 'Starting / Partindo';
                vfdStartCmd := TRUE;
                tonRunFbWait(IN := TRUE, PT := vfdRunFbTimeout);
                step := 10;
            END_IF
        END_IF

    // ========================== 10) STARTING ==========================
    10:
        running     := FALSE;
        vfdStartCmd := TRUE;
        deviceState := 'Starting (await RUN fb) / Aguardando RUN';

        // Falha ou perda de condição => parar
        IF vfdFaultFeedback THEN
            faultActive := TRUE;
            faultMsg := 'Fault from VFD';
            vfdStartCmd := FALSE;
            tonRunFbWait(IN := FALSE);
            runLatch := FALSE;
            step := 90;

        ELSIF NOT vfdReady THEN
            deviceState := 'Stopping: VFD not ready / Parando: inversor NOK';
            vfdStartCmd := FALSE;
            tonRunFbWait(IN := FALSE);
            runLatch := FALSE;
            step := 90;

        // Interlocks em START: classe normal (parada)
        ELSIF NOT allInterlocksOK THEN
            deviceState := 'Stopping: interlock open / Parando: intertravamento';
            vfdStartCmd := FALSE;
            tonRunFbWait(IN := FALSE);
            runLatch := FALSE;
            step := 90;

        // Chegou RUN?
        ELSIF vfdRunFeedback THEN
            tonRunFbWait(IN := FALSE);
            step := 20;

        // Timeout?
        ELSIF tonRunFbWait.Q THEN
            faultActive := TRUE;
            faultMsg := 'Start failed: RUN fb timeout / Falha partida: tempo RUN';
            deviceState := faultMsg;
            vfdStartCmd := FALSE;
            tonRunFbWait(IN := FALSE);
            runLatch := FALSE;
            step := 90;
        END_IF

    // =========================== 20) RUNNING ===========================
    20:
        running     := TRUE;           // libera intertravamento de outros grupos
        vfdStartCmd := TRUE;
        deviceState := 'Running / Operando';

        // Supervisão contínua
        IF vfdFaultFeedback THEN
            faultActive := TRUE;
            faultMsg := 'Fault from VFD';
            vfdStartCmd := FALSE;
            runLatch := FALSE;
            step := 90;

        ELSIF NOT vfdReady THEN
            deviceState := 'Stopping: VFD not ready';
            vfdStartCmd := FALSE;
            runLatch := FALSE;
            step := 90;

        ELSIF NOT vfdRunFeedback THEN
            deviceState := 'Stopping: RUN feedback lost';
            vfdStartCmd := FALSE;
            runLatch := FALSE;
            step := 90;

        // Interlocks: parada normal
        ELSIF NOT allInterlocksOK THEN
            deviceState := 'Stopping: interlock open';
            vfdStartCmd := FALSE;
            runLatch := FALSE;
            step := 90;

        // Start foi destoggleado (runLatch caiu)?
        ELSIF NOT runLatch THEN
            deviceState := 'Stopping (Start toggled off) / Parando (Start OFF)';
            vfdStartCmd := FALSE;
            step := 90;

        ELSE
            // ================== LOOP DE CONTROLE (ativo em RUN) ==================
            // 1) Ajuste de razão por botões (mantido do original)
            _SetpointInputControl();

            // 2) Jet-to-wire → SP automático [mmH2O]
            _JetToWire(
                wireSpeedMPM        := formingBoardSpeedMPM,
                ratio               := jetToWireRatio,
                gainK               := jetHeadGainK,
                offset_mmH2O        := jetHeadOffset_mmH2O,
                minSP_mmH2O         := minAutoSP_mmH2O,
                maxSP_mmH2O         := maxAutoSP_mmH2O,
                jetSpeed_mps        => jetSpeed_mps,
                autoSetpoint_mmH2O  => headBoxMMH2OCalc
            );

            // 3) Filtro PT1 da PV (habilitável)
            _InputFilter(
                enableFilter  := enableInputFilter,
                rawValue      := pressureFeedback_mmH2O,
                filterTime    := inputFilterTime,
                filterGainK   := inputFilterGainK,
                filteredValue => filteredPV_mmH2O
            );
            // headBoxMMH2ORead é atualizado dentro de _InputFilter (mantido)

            // 4) Manual clamp
            manualCmdPct := LIMIT(outLowLimitPct, manualSetpoint, outHighLimitPct);

            // 5) PID OSCAT (ACT/SET em mmH2O, Y em %)
            instPID(
                ACT := filteredPV_mmH2O,
                SET := headBoxMMH2OCalc,
                SUP := pidDeadband_mmH2O,
                OFS := outputOffsetPct,
                M_I := manualCmdPct,
                MAN := NOT autoMode,
                RST := resetPID,
                KP  := kp,
                TN  := tn,
                TV  := tv,

                Y   => yPID_Pct,
                DIFF=> pidDiff,
                LIM => pidLimited
            );

            // 6) Seleção modo & clamp final da referência do VFD
            IF autoMode THEN
             vfdSpeedPct := yPID_Pct;
			 //vfdSpeedPct := manualCmdPct;
             instPID.LL  := outLowLimitPct;
             instPID.LH  := outHighLimitPct;		 
			 
  
            ELSE
				
                vfdSpeedPct := manualCmdPct;
				instPID.LL  := manualCmdPct;
				instPID.LH  := manualCmdPct;	
			
            END_IF
			
			
			IF instTON_RunningDelay.Q THEN
			
				vfdSpeedPct := LIMIT(outLowLimitPct, vfdSpeedPct, outHighLimitPct);

			ELSE
				
				vfdSpeedPct := LIMIT(5, vfdSpeedPct, 10.0);

			END_IF
			
			
			
        END_IF

    // =========================== 90) STOPPING ==========================
    90:
        running     := FALSE;
        vfdStartCmd := FALSE;
        vfdSpeedPct := 0.0;
        tonRunFbWait(IN := FALSE);
        deviceState := 'Stopping / Parando';

        // Retorna a IDLE quando liberar stop e condições estiverem OK
        IF NOT stopCommand THEN
            step := 0; // Idle
        END_IF

    // ============================ DEFAULT =============================
    ELSE
        running     := FALSE;
        vfdStartCmd := FALSE;
        vfdSpeedPct := 0.0;
        tonRunFbWait(IN := FALSE);
        step := 0;
END_CASE;

// --------------------- Displays (corrente/torque) ---------------------
_FeedbackDisplay();


instTON_RunningDelay(IN:= running, PT := T#40S);

METHOD _FeedbackDisplay
VAR_INPUT
END_VAR
VAR CONSTANT
    STATUS_IDLE     : INT := 0;
//    STATUS_STARTING : INT := 1;
    STATUS_RUNNING  : INT := 1;
    STATUS_FAULT    : INT := 2;
END_VAR
// ───────────────────────── 5) HMI DISPLAY SIGNALS ─────────────────────────────
// Filtered speed for HMI (Velocidade filtrada para HMI)
instPT1_SpeedDisplay(
    in  := vfdEngFeedback,             // raw speed feedback (velocidade bruta)
    T   := displayFilterTime,          // small smoothing (suavização leve)
    K   := 1.0,
    out => vfdEngDisplay               // speed shown on HMI (velocidade na HMI)
);

// Filtered torque for HMI (Torque filtrado para HMI)
instPT1_TorqueDisplay(
    in  := vfdTorqueFeedback,          // raw torque (torque bruto)
    T   := displayFilterTime,
    K   := 1.0,
    out => vfdTorqueDisplay            // torque shown on HMI (torque na HMI)
);

// Filtered current for HMI (Corrente filtrada para HMI)
instPT1_CurrentDisplay(
    in  := vfdCurrentFeedback,         // raw current (corrente bruta)
    T   := displayFilterTime,
    K   := 1.0,
    out => vfdCurrentDisplay           // current shown on HMI (corrente na HMI)
);

// ───────────────────────── GROUP STATUS / STATUS CODE ─────────────────────────
// 0=Idle, 1=Starting, 2=Running, 3=Fault  (códigos para HMI)
IF vfdFaultFeedback OR faultActive THEN
    statusCode := STATUS_FAULT;         // Fault (Falha)
ELSIF vfdRunFeedback THEN
    statusCode := STATUS_RUNNING;         // Running (Operando)
ELSE
    statusCode := STATUS_IDLE;         // Idle (Parado)
END_IF;


(*

// Master drive
IF masterVfdFaultFeedback THEN
    masterStatusCode := STATUS_FAULT;
ELSIF masterVfdRunFeedback THEN
    masterStatusCode := STATUS_RUNNING;
ELSE
    masterStatusCode := STATUS_IDLE;
END_IF;

// Slave drive
IF slaveVfdFaultFeedback THEN
    slaveStatusCode := STATUS_FAULT;
ELSIF slaveVfdRunFeedback THEN
    slaveStatusCode := STATUS_RUNNING;
ELSE
    slaveStatusCode := STATUS_IDLE;
END_IF;

*)
END_METHOD

// ============================================================================
// METHOD: _InputFilter
// OSCAT PT1 filter for PV, with enable/disable and bumpless behavior.
// When disabled, the filter tracks input quickly (tiny T) to avoid bumps.
// ============================================================================
METHOD PRIVATE _InputFilter
VAR_INPUT
    enableFilter   : BOOL;  // TRUE=apply PT1, FALSE=bypass
    rawValue       : REAL;  // Input value to be filtered
    filterTime     : TIME;  // PT1 time constant
    filterGainK    : REAL;  // PT1 gain, typically 1.0
END_VAR
VAR_OUTPUT
    filteredValue  : REAL;  // Filtered (or bypassed) value
END_VAR
VAR
    kUse           : REAL;
    tUse           : TIME;
    yPT1           : REAL;
END_VAR


IF enableFilter THEN
    kUse := filterGainK;
    tUse := filterTime;
ELSE
    // Track input closely for bumpless re-enable
    kUse := 1.0;
    tUse := T#10ms;
END_IF;

instsFT_PT1TInputFilter(
    in  := rawValue,
//    T   := tUse,
    T   := T#8s,

    K   := kUse,
    out => yPT1
);

// Output selection
IF enableFilter THEN
    filteredValue := yPT1;
ELSE
    filteredValue := rawValue;
END_IF;

//Display filtered value output
headBoxMMH2ORead := yPT1;
END_METHOD

// ============================================================================
// METHOD: _JetToWire
// Computes jet speed from wire speed and ratio, then maps to pressure SP (mmH2O).
// Dynamic head: H[mmH2O] = (v^2 / (2*g)) * 1000, with g = 9.80665 m/s^2.
// A tunable gain/offset is applied; SP is clamped to min/max bounds.
// ============================================================================
METHOD PRIVATE _JetToWire
VAR_INPUT
    wireSpeedMPM        : REAL;  // Wire speed [m/min]
    ratio               : REAL;  // Jet/Wire ratio (unitless), e.g., 1.05
    gainK               : REAL;  // Gain on computed head
    offset_mmH2O        : REAL;  // Offset added to head [mmH2O]
    minSP_mmH2O         : REAL;  // SP lower bound [mmH2O]
    maxSP_mmH2O         : REAL;  // SP upper bound [mmH2O]
END_VAR
VAR_OUTPUT
    jetSpeed_mps        : REAL;  // Jet speed [m/s]
    autoSetpoint_mmH2O  : REAL;  // Pressure SP [mmH2O]
END_VAR
VAR
    wire_mps            : REAL;
    rUse                : REAL;
    dynHead_mmH2O       : REAL;
    cHeadCoeff          : REAL := 50.988; // 1000/(2*g), g=9.80665
END_VAR
// Sanitize ratio
rUse := ratio;
IF rUse < 0.0 THEN rUse := 0.0; END_IF;

// Convert wire speed to m/s
wire_mps := wireSpeedMPM / 60.0;

// Jet speed and dynamic head
jetSpeed_mps := rUse * wire_mps;
dynHead_mmH2O := cHeadCoeff * (jetSpeed_mps * jetSpeed_mps);

// Apply gain/offset and clamp
autoSetpoint_mmH2O := gainK * dynHead_mmH2O + offset_mmH2O;
IF autoSetpoint_mmH2O < minSP_mmH2O THEN autoSetpoint_mmH2O := minSP_mmH2O; END_IF;
IF autoSetpoint_mmH2O > maxSP_mmH2O THEN autoSetpoint_mmH2O := maxSP_mmH2O; END_IF;
END_METHOD

// ============================================================================
// METHOD: _SetpointInputControl
// Purpose: Handle HMI writes and button nudges for both ratio and manual SP,
//          using OSCAT TUNE2 instances. External writes trigger a one-scan
//          SET pulse; SU/SD remain active every scan.
// Objetivo: Tratar escritas da HMI e botões ↑/↓ para razão e SP manual,
//           usando TUNE2. Escritas externas disparam SET por 1 varredura;
//           SU/SD permanecem ativos a cada ciclo.
// ============================================================================

METHOD PRIVATE _SetpointInputControl

// ─────────────────────────── Jet-to-Wire Ratio (Razão) ─────────────────────────
// External change detection: if HMI/ADS writes a value larger than the step,
// pulse SET to push it into TUNE2.
// Detecção de mudança externa: se HMI/ADS gravar valor maior que o passo,
// pulsar SET para aplicar no TUNE2.
IF ABS(jetToWireRatio - jetToWireRatioOld) > instTUNE2RatioSetpoint.SS THEN
    // Clamp to tuner limits (garante limites)
    // One-scan SET pulse to sync internal setpoint (pulso SET de 1 ciclo)
    instTUNE2RatioSetpoint(
        SET_val := jetToWireRatio,
        SET     := TRUE
    );
    instTUNE2RatioSetpoint(SET := FALSE);

    // Remember applied value (memoriza valor aplicado)
END_IF;

// Track last seen value (rastreia último valor observado)
jetToWireRatioOld := jetToWireRatio;

// Normal SU/SD operation (operação normal dos botões ↑/↓)
instTUNE2RatioSetpoint(
    SET      := FALSE,               // No direct set here (sem SET contínuo)
    SU       := jetToWireRatioInc,   // Increment button (↑)
    SD       := jetToWireRatioDec,   // Decrement button (↓)
    RST      := FALSE,               // Optional external reset (reset opcional)
    SS       := jetToWireRatioStep,  // Small step per press (passo fino)
    FS       := 0.0,                 // Fast step (unused) (passo rápido, não usado)
    LIMIT_L  := jetToWireRatioMin,   // Lower bound (limite inferior)
    LIMIT_H  := jetToWireRatioMax,   // Upper bound (limite superior)
    Y        => jetToWireRatio       // Current ratio output (saída da razão)
);


// ─────────────────────────── Manual Setpoint (SP Manual) ───────────────────────
// Same pattern: detect external write > step, pulse SET, then keep SU/SD active.
// Mesmo padrão: detectar escrita externa > passo, pulsar SET, manter SU/SD ativo.
IF ABS(manualSetpoint - manualSetpointOld) > instTUNE2ManSetpoint.SS THEN
    // Clamp to tuner limits (garante limites)
    // One-scan SET pulse to sync internal setpoint (pulso SET de 1 ciclo)
    instTUNE2ManSetpoint(
        SET_val := manualSetpoint,
        SET     := TRUE
    );
    instTUNE2ManSetpoint(SET := FALSE);

    // Remember applied value (memoriza valor aplicado)
END_IF;

// Track last seen value (rastreia último valor observado)
manualSetpointOld := manualSetpoint;

// Normal SU/SD operation (operação normal dos botões ↑/↓)
instTUNE2ManSetpoint(
    SET      := FALSE,               // No direct set here (sem SET contínuo)
    SU       := manualSetpointInc,   // Increment button (↑)
    SD       := manualSetpointDec,   // Decrement button (↓)
    RST      := FALSE,               // Optional external reset (reset opcional)
    SS       := 0.1,                 // Small step per press (passo fino)
    FS       := 0.0,                 // Fast step (unused) (passo rápido, não usado)
    LIMIT_L  := 0.0,                 // Lower bound (limite inferior)
    LIMIT_H  := 100,                 // Upper bound (limite superior)
    Y        => manualSetpoint       // Current manual SP output (saída do SP manual)
);
END_METHOD

END_FUNCTION_BLOCK

// ---- Function Blocks/PaperMachine/Auxiliary/FB_VfdProcessControler.TcPOU
(*
    FB_ProcessControler
    Purpose: Generic process controller with start/stop latch, status codes,
             PID (OSCAT CTRL_PID), optional reverse action, PV PT1 filter,
             engineering↔% scaling, drive run supervision, and HMI displays.

    Sequence: Start pulse toggles RUN latch; Stop pulse/level forces stop.

    Status codes: statusCode INT → 0=Idle, 1=Running, 2=Fault

    Notes: Includes optional low/high PV “hold” with hysteresis (normal-stop class).
*)

FUNCTION_BLOCK FB_VfdProcessControler
VAR_INPUT
    // ===== Sequence commands =====
    startCommand                 : BOOL;            // Start pulse toggles RUN latch
    stopCommand                  : BOOL;            // Stop pulse/level forces stop

    // ===== Manual output & Auto SP nudge =====
    processSetpointManInc        : BOOL;            // Manual output ↑ (0..100%)
    processSetpointManDec        : BOOL;            // Manual output ↓ (0..100%)
    processSetpointManSteps      : REAL := 0.1;

    processSetpointAutoInc       : BOOL;            // Auto SP ↑ (engineering units or %)
    processSetpointAutoDec       : BOOL;            // Auto SP ↓ (engineering units or %)
    processSetpointAutoSteps     : REAL := 1.0;

    // ===== Mode =====
    autoMode                     : BOOL;            // TRUE=Automatic / FALSE=Manual
    reverseActing                : BOOL := FALSE;   // TRUE: higher output decreases PV; FALSE: direct

    // ===== Process signals (PV in engineering units) =====
    processFeedbackEng           : REAL;            // PV (engineering units), e.g., bar/kPa/°C/…

    // ===== PID parameters (OSCAT CTRL_PID) =====
    kp                           : REAL := 1.0;     // Proportional gain (sign handled via reverseActing)
    tn                           : REAL := 8.0;     // Integral time [s]
    tv                           : REAL := 0.0;     // Derivative time [s]

    // ===== Output limits & offset =====
    outLowLimitPct               : REAL := 0.0;     // Min output %
    outHighLimitPct              : REAL := 100.0;   // Max output %
    outputOffsetPct              : REAL := 0.0;     // Offset added to final output

    // ===== PID housekeeping =====
    resetPID                     : BOOL;            // Reset integrator

    // ===== Input filter (OSCAT FT_PT1) =====
    enableInputFilter            : BOOL := TRUE;    // Enable PV PT1 filter
    inputFilterTime              : TIME := T#300ms; // PT1 time constant
    inputFilterGainK             : REAL := 1.0;     // PT1 gain

    displayFilterTime            : TIME := T#20ms;  // Small PT1 for HMI displays

    // ===== Optional scaling (engineering ↔ %) =====
    enableScaling                : BOOL := TRUE;    // Enable engineering↔% scaling
    pLoEng                       : REAL := 0.0;     // Engineering low bound
    pHiEng                       : REAL := 10.0;    // Engineering high bound

    // ===== Drive interface & supervision (VFD or actuator drive) =====
    vfdReady                     : BOOL;            // Drive ready/healthy
    vfdRunFeedback               : BOOL;            // Drive RUN feedback
    vfdFaultFeedback             : BOOL;            // Drive fault
    vfdRunFbTimeout              : TIME := T#5s;    // Timeout to receive RUN FB after start

    // ===== Drive analog feedbacks (for HMI display) =====
    vfdCurrentFeedback           : REAL;            // Current [A or %]
    vfdEngFeedback               : REAL;            // Engineering feedback (e.g., rpm, flow, etc.)
    vfdTorqueFeedback            : REAL;            // Torque (Nm or %)

    // ===== Safety (true safety inputs only) =====
    safetyOk                     : BOOL := TRUE;    // Safety chain OK
    estopOk                      : BOOL := TRUE;    // E-Stop loop OK
    guardClosedOk                : BOOL := TRUE;    // Guards/doors closed

    // ===== Interlocks (process permissives) — normal stop only =====
    interlock1                   : BOOL := TRUE;
    interlock2                   : BOOL := TRUE;
    interlock3                   : BOOL := TRUE;
    interlock4                   : BOOL := TRUE;
    interlock5                   : BOOL := TRUE;
    interlock6                   : BOOL := TRUE;

 // ===== Optional low-PV hold (normal-stop/hold) =====
    minPVEnable                  : BOOL := FALSE;   // Enable low-PV hold
    minPVTripEng                 : REAL := 0.5;     // Trip threshold (engineering units)
    minPVReleaseEng              : REAL := 0.7;     // Release threshold (engineering units)
    minPVTripTime                : TIME := T#1s;    // PV < trip for this long to trip
    minPVReleaseTime             : TIME := T#1s;    // PV > release for this long to release

    // ===== Optional high-PV hold (normal-stop/hold) =====
    maxPVEnable                  : BOOL := FALSE;   // Enable high-PV hold
    maxPVTripEng                 : REAL := 9.5;     // Trip threshold (engineering units)
    maxPVReleaseEng              : REAL := 9.2;     // Release threshold (engineering units)
    maxPVTripTime                : TIME := T#1s;    // PV > trip for this long to trip
    maxPVReleaseTime             : TIME := T#1s;    // PV < release for this long to release
	
	
END_VAR

VAR_OUTPUT
    running                      : BOOL;            // TRUE only during RUN state
    controlOutputPct             : REAL;            // Final control output 0..100%
    pidDiff                      : REAL;            // SET − ACT (post-scaling)
    pidLimited                   : BOOL;            // TRUE if saturated
    deviceState                  : STRING(80);      // Human-readable state
    vfdStartCmdOut               : BOOL;            // Asserted in Start/Run to the drive

    // ===== Holds (normal stop class) =====
    minPressureHoldActive        : BOOL;            // Low-PV hold active
    maxPressureHoldActive        : BOOL;            // High-PV hold active

    // ===== Status & HMI displays =====
    statusCode                   : INT;             // 0=Idle, 1=Running, 2=Fault
    vfdCurrentDisplay            : REAL;            // Display current [A or %]
    vfdTorqueDisplay             : REAL;            // Display torque (Nm or %)
    vfdEngDisplay                : REAL;            // Display engineering feedback (e.g., rpm)
    processFeedbackEngDisplay    : REAL;            // PV (engineering units), e.g., bar/kPa/°C/…
	
	
END_VAR

VAR
    // ===== First scan & state/edges =====
    firstScan                    : BOOL := TRUE;    // TRUE only on first PLC cycle

    step                         : INT;             // 0=Idle,10=Starting,20=Running,90=Stopping
    startOld                     : BOOL;            // Edge memory
    stopOld                      : BOOL;            // Edge memory
    rStart                       : BOOL;            // Rising edge: start
    rStop                        : BOOL;            // Rising edge: stop
    runLatch                     : BOOL;            // Toggled by Start; cleared by Stop

    // ===== Internals =====
    manualCmd                    : REAL;            // Manual command %
    yPID                         : REAL;            // PID output %
    kpUse                        : REAL;            // Kp adjusted by reverseActing

    // ===== Filtered PV (engineering units) =====
    pvEngFiltered                : REAL;

    // ===== PV & SP in % (post-scaling) =====
    pvPct                        : REAL;
    spPct                        : REAL;

    // ===== Timers =====
    tonRunFbWait                 : TON;             // Waits RUN FB after start

    // ===== Low/High PV timers =====
    tonMinPTrip                  : TON;
    tonMinPRelease               : TON;
    tonMaxPTrip                  : TON;
    tonMaxPRelease               : TON;

    // ===== Instances =====
    instPID                      : CTRL_PID;        // OSCAT PID
    instPT1                      : FT_PT1;          // PV PT1 filter

    // ===== Aggregations =====
    allSafetyOK                  : BOOL;            // safetyOk & estopOk & guardClosedOk
    anyInterlockOpen             : BOOL;            // any interlock is FALSE

    // ===== HMI display filters =====
    instPT1_TorqueDisplay        : FT_PT1;          // PT1 for torque display
    instPT1_SpeedDisplay         : FT_PT1;          // PT1 for engineering display
    instPT1_ProcessFeedbackEngDisplay        : FT_PT1;          // PT1 for engineering display
	

    processSetpointManOld        : REAL;            // Last observed manual SP (HMI)
    processSetpointAutoOld       : REAL;            // Last observed auto SP (HMI)
	minPVHoldActive: BOOL;
	maxPVHoldActive: BOOL;
END_VAR

VAR PERSISTENT
    instTUNE2AutoSetpoint        : TUNE2;           // OSCAT TUNE2 for auto SP nudge
    instTUNE2ManSetpoint         : TUNE2;           // OSCAT TUNE2 for manual output
END_VAR

VAR_IN_OUT
    // ===== Exposed setpoints =====
    processSetpointMan           : REAL;            // Manual output 0..100%
    processSetpointAuto          : REAL;            // Auto SP (engineering units or % per configuration)
END_VAR

// ============================ INITIALIZATION ============================
// Run this block only once on first cycle
IF firstScan THEN
    firstScan := FALSE;

    processSetpointMan      := instTUNE2ManSetpoint.Y;
    processSetpointManOld   := processSetpointMan;

    processSetpointAuto     := instTUNE2AutoSetpoint.Y;
    processSetpointAutoOld  := processSetpointAuto;
END_IF;


// ============================ Edges ============================
rStart := startCommand AND NOT startOld;
startOld := startCommand;

rStop  := stopCommand AND NOT stopOld;
stopOld := stopCommand;

// Start toggles run; Stop forces stop
IF rStart THEN
    runLatch := TRUE;
END_IF;
IF rStop OR stopCommand THEN
    runLatch := FALSE;
END_IF;


// ============================ Aggregations =====================
allSafetyOK := safetyOk AND estopOk AND guardClosedOk;
anyInterlockOpen := NOT (interlock1 AND interlock2 AND interlock3 AND interlock4 AND interlock5 AND interlock6);

// Defaults each cycle
vfdStartCmdOut := FALSE;


// ============================ Low/High PV HOLD supervision ============================
// LOW-PV
IF minPVEnable THEN
    tonMinPTrip   (IN := (processFeedbackEng <  minPVTripEng),     PT := minPVTripTime);
    tonMinPRelease(IN := (processFeedbackEng >  minPVReleaseEng),  PT := minPVReleaseTime);
    IF tonMinPTrip.Q    THEN minPVHoldActive := TRUE;  END_IF;
    IF tonMinPRelease.Q THEN minPVHoldActive := FALSE; END_IF;
	
ELSE
    tonMinPTrip(IN := FALSE);
    tonMinPRelease(IN := FALSE);
    minPVHoldActive := FALSE;
END_IF;

// HIGH-PV
IF maxPVEnable THEN
    tonMaxPTrip   (IN := (processFeedbackEng > maxPVTripEng),       PT := maxPVTripTime);
    tonMaxPRelease(IN := (processFeedbackEng < maxPVReleaseEng),    PT := maxPVReleaseTime);
    IF tonMaxPTrip.Q    THEN maxPVHoldActive := TRUE;  END_IF;
    IF tonMaxPRelease.Q THEN maxPVHoldActive := FALSE; END_IF;
	
ELSE
    tonMaxPTrip(IN := FALSE);
    tonMaxPRelease(IN := FALSE);
    maxPVHoldActive := FALSE;
END_IF;


// ============================ Immediate stop / safety/fault =================
IF rStop OR stopCommand THEN
    controlOutputPct := 0.0;
    running := FALSE;
    deviceState := 'Stopping (Stop command)';
    runLatch := FALSE;
    step := 90;
END_IF;

IF vfdFaultFeedback THEN
    deviceState := 'Fault from drive';
    runLatch := FALSE;
    step := 90;
END_IF;

IF NOT allSafetyOK THEN
    deviceState := 'Stopping: safety chain open';
    runLatch := FALSE;
    step := 90;
END_IF;


// ============================ State machine =====================
CASE step OF
    // ------------------------------------------------------------
    0: // Idle
        running := FALSE;
        controlOutputPct := 0.0;
        deviceState := 'Idle';
        vfdStartCmdOut := FALSE;

        // Start request via runLatch (toggled by Start pulse)
        IF runLatch AND NOT stopCommand THEN
            // Safety must be OK; drive must be ready; holds must be clear
            IF NOT allSafetyOK THEN
                deviceState := 'Start blocked: safety not OK';
                runLatch := FALSE;
                step := 0;
            ELSIF NOT vfdReady THEN
                deviceState := 'Start blocked: drive not ready';
                runLatch := FALSE;
                step := 0;
            ELSIF (minPVEnable AND minPVHoldActive) OR (maxPVEnable AND maxPVHoldActive) THEN
                deviceState := 'Start blocked: PV hold active';
                runLatch := FALSE;
                step := 0;
            ELSE
                deviceState := 'Starting';
                vfdStartCmdOut := TRUE;                   // send START to drive
                tonRunFbWait(IN := TRUE, PT := vfdRunFbTimeout);
                step := 10;
            END_IF
        END_IF

    // ------------------------------------------------------------
    10: // Starting (await RUN feedback)
        running := FALSE;
        deviceState := 'Starting (await RUN feedback)';
        vfdStartCmdOut := TRUE;

        // Safety/fault during start => stop
        IF NOT allSafetyOK THEN
            tonRunFbWait(IN := FALSE);
            deviceState := 'Stopping: safety chain open';
            vfdStartCmdOut := FALSE;
            runLatch := FALSE;
            step := 90;

        ELSIF vfdFaultFeedback THEN
            tonRunFbWait(IN := FALSE);
            deviceState := 'Fault from drive';
            vfdStartCmdOut := FALSE;
            runLatch := FALSE;
            step := 90;

        // Interlocks are normal stop only
        ELSIF anyInterlockOpen THEN
            tonRunFbWait(IN := FALSE);
            deviceState := 'Stopping: interlock open';
            vfdStartCmdOut := FALSE;
            runLatch := FALSE;
            step := 90;

        // PV holds => normal stop
        ELSIF (minPVEnable AND minPVHoldActive) OR (maxPVEnable AND maxPVHoldActive) THEN
            tonRunFbWait(IN := FALSE);
            deviceState := 'Stopping: PV hold';
            vfdStartCmdOut := FALSE;
            runLatch := FALSE;
            step := 90;

        // RUN feedback arrived
        ELSIF vfdRunFeedback THEN
            tonRunFbWait(IN := FALSE);
            step := 20;

        // Timeout
        ELSIF tonRunFbWait.Q THEN
            tonRunFbWait(IN := FALSE);
            deviceState := 'Start failed: RUN feedback timeout';
            vfdStartCmdOut := FALSE;
            runLatch := FALSE;
            step := 90;
        END_IF

    // ------------------------------------------------------------
    20: // Running (control loop)
        running := TRUE;               // may be used to release other devices
        deviceState := 'Running';
        vfdStartCmdOut := TRUE;

        // Supervision
        IF NOT allSafetyOK THEN
            deviceState := 'Stopping: safety chain open';
            vfdStartCmdOut := FALSE;
            runLatch := FALSE;
            step := 90;

        ELSIF vfdFaultFeedback THEN
            deviceState := 'Fault from drive';
            vfdStartCmdOut := FALSE;
            runLatch := FALSE;
            step := 90;

        ELSIF NOT vfdReady THEN
            deviceState := 'Stopping: drive not ready';
            vfdStartCmdOut := FALSE;
            runLatch := FALSE;
            step := 90;

        ELSIF NOT vfdRunFeedback THEN
            deviceState := 'Stopping: RUN feedback lost';
            vfdStartCmdOut := FALSE;
            runLatch := FALSE;
            step := 90;

        // Interlocks → normal stop
        ELSIF anyInterlockOpen THEN
            deviceState := 'Stopping: interlock open';
            vfdStartCmdOut := FALSE;
            runLatch := FALSE;
            step := 90;

        // PV holds → normal stop
        ELSIF (minPVEnable AND minPVHoldActive) OR (maxPVEnable AND maxPVHoldActive) THEN
            deviceState := 'Stopping: PV hold';
            vfdStartCmdOut := FALSE;
            runLatch := FALSE;
            step := 90;

        // Start toggled OFF while running => stop
        ELSIF NOT runLatch THEN
            deviceState := 'Stopping (Start toggled off)';
            vfdStartCmdOut := FALSE;
            step := 90;

        ELSE
            // ---- Input filtering (PT1) ----
            IF enableInputFilter THEN
                instPT1(in := processFeedbackEng, T := inputFilterTime, K := inputFilterGainK, out => pvEngFiltered);
            ELSE
                pvEngFiltered := processFeedbackEng;
            END_IF

            // ---- Engineering → % scaling ----
            IF enableScaling THEN
                pvPct := _ScaleToPct(pvEngFiltered,       pLoEng, pHiEng);
                spPct := _ScaleToPct(processSetpointAuto, pLoEng, pHiEng);
            ELSE
                pvPct := pvEngFiltered;        // already %
                spPct := processSetpointAuto;  // already %
            END_IF

            // ---- Manual path and PID with bumpless transfer ----
            manualCmd := LIMIT(0.0, processSetpointMan, 100.0);

            // Reverse/direct action by Kp sign
            IF reverseActing THEN
                kpUse := -ABS(kp);
            ELSE
                kpUse :=  ABS(kp);
            END_IF

            instPID(
                ACT := pvPct,
                SET := spPct,
                M_I := manualCmd,
                MAN := NOT autoMode,
                RST := resetPID,
                KP  := kpUse,
                TN  := tn,
                TV  := tv,
                LL  := outLowLimitPct,
                LH  := outHighLimitPct,
                Y   => yPID,
                DIFF=> pidDiff,
                LIM => pidLimited
            );

            // Mode select, offset, clamp
            IF autoMode THEN
                controlOutputPct := yPID;
            ELSE
                controlOutputPct := manualCmd;
            END_IF
            controlOutputPct := LIMIT(outLowLimitPct, controlOutputPct + outputOffsetPct, outHighLimitPct);
        END_IF

    // ------------------------------------------------------------
    90: // Stopping (normal, de-energize)
        running := FALSE;
        controlOutputPct := 0.0;
        vfdStartCmdOut := FALSE;
        tonRunFbWait(IN := FALSE);

        // Return to Idle once stop released and safety OK
        IF NOT stopCommand AND allSafetyOK THEN
            deviceState := 'Idle';
            step := 0;
        END_IF

    // ------------------------------------------------------------
    ELSE
        running := FALSE;
        controlOutputPct := 0.0;
        deviceState := 'Idle';
        vfdStartCmdOut := FALSE;
        step := 0;
END_CASE;


// =============================== Status code ===============================
IF vfdFaultFeedback THEN
    statusCode := 2;             // Fault
ELSIF running THEN
    statusCode := 1;             // Running
ELSE
    statusCode := 0;             // Idle
END_IF

// HMI feedbacks & status (encapsulates PT1 displays and status code if desired)
_FeedbackDisplay();

// Setpoint input handling (encapsulates TUNE2-based HMI writes & nudges)
_SetpointInputControl();

METHOD _FeedbackDisplay
VAR_INPUT
END_VAR
// 5) HMI DISPLAY SIGNALS (filtered speeds/torques + GROUP status)
instPT1_SpeedDisplay(in := vfdEngFeedback, T := displayFilterTime, K := 1.0, out => vfdEngDisplay);
instPT1_TorqueDisplay (in := vfdTorqueFeedback , T := displayFilterTime, K := 1.0, out => vfdTorqueDisplay);
instPT1_ProcessFeedbackEngDisplay(in := processFeedbackEng , T := displayFilterTime, K := 1.0, out => processFeedbackEngDisplay);
END_METHOD

// ============================ Helper ============================
METHOD PRIVATE _ScaleToPct : REAL
VAR_INPUT
    xEng  : REAL;  // value in engineering units
    loEng : REAL;  // min eng
    hiEng : REAL;  // max eng
END_VAR
VAR
    span : REAL;
    pct  : REAL;
END_VAR

span := hiEng - loEng;
IF span = 0.0 THEN
    _ScaleToPct := 0.0; // avoid div by zero
ELSE
    pct := (xEng - loEng) / span * 100.0;
    _ScaleToPct := LIMIT(0.0, pct, 100.0);
END_IF
END_METHOD

// ============================================================================
// METHOD: _SetpointInputControl
// Purpose: Handle HMI writes for manual output using OSCAT TUNE2. Any external
//          write to manualOutputPct bigger than the configured step will pulse
//          SET for one scan. No SU/SD buttons here (PressureCtrl doesn’t use them).
// Objetivo: Tratar escrita da HMI no manualOutputPct via TUNE2. Mudança externa
//           > passo gera pulso SET de 1 varredura. Sem botões ↑/↓ neste FB.
// ============================================================================
METHOD PRIVATE _SetpointInputControl
VAR
    spManClamped : REAL;
    spAutoClamped : REAL;
	
END_VAR
// Detect external write (> step): ignore tiny jitter
IF ABS(processSetpointMan - processSetpointManOld) > instTUNE2ManSetpoint.SS THEN
    // Clamp to output limits before writing (garante limites)
    spManClamped := LIMIT(outLowLimitPct, processSetpointMan, outHighLimitPct);

    // One-scan SET pulse into TUNE2 (pulso SET de 1 ciclo)
    instTUNE2ManSetpoint(
        SET_val := spManClamped,
        SET     := TRUE
    );
    instTUNE2ManSetpoint(SET := FALSE);

    // Remember applied value (memoriza)
    processSetpointManOld := processSetpointMan;
ELSE
    // Track last seen to avoid drift (rastreia último observado)
    processSetpointManOld := processSetpointMan;
END_IF;

// Keep TUNE2 active (no SU/SD in this FB)
instTUNE2ManSetpoint(
    SET      := FALSE,
    SU       := processSetpointManInc,
    SD       := processSetpointManDec,
    RST      := FALSE,
    SS       := 0.1,           // step reference (passo de referência)
    FS       := 0.0,                     // unused
    LIMIT_L  := outLowLimitPct,
    LIMIT_H  := outHighLimitPct,
    Y        => processSetpointMan
);




// Detect external write (> step): ignore tiny jitter
IF ABS(processSetpointAuto - processSetpointAutoOld) > instTUNE2AutoSetpoint.SS THEN
    // Clamp to output limits before writing (garante limites)
    spAutoClamped := LIMIT(0, processSetpointAuto, 100);

    // One-scan SET pulse into TUNE2 (pulso SET de 1 ciclo)
    instTUNE2AutoSetpoint(
        SET_val := spAutoClamped,
        SET     := TRUE
    );
    instTUNE2AutoSetpoint(SET := FALSE);

    // Remember applied value (memoriza)
    processSetpointAutoOld := processSetpointAuto;
ELSE
    // Track last seen to avoid drift (rastreia último observado)
    processSetpointAutoOld := processSetpointAuto;
END_IF;

// Keep TUNE2 active (no SU/SD in this FB)
instTUNE2AutoSetpoint(
    SET      := FALSE,
    SU       := processSetpointAutoInc,
    SD       := processSetpointAutoDec,
    RST      := FALSE,
    SS       := 0.1,           // step reference (passo de referência)
    FS       := 0.0,                     // unused
    LIMIT_L  := 0.0,
    LIMIT_H  := 100.0,
    Y        => processSetpointAuto
);
END_METHOD

END_FUNCTION_BLOCK

// ---- Function Blocks/PaperMachine/Auxiliary/FB_WirePitControl.TcPOU
(*
    FB_ProcessControler
    Purpose: Generic process controller with start/stop latch, status codes,
             PID (OSCAT CTRL_PID), optional reverse action, PV PT1 filter,
             engineering↔% scaling, drive run supervision, and HMI displays.

    Sequence: Start pulse toggles RUN latch; Stop pulse/level forces stop.

    Status codes: statusCode INT → 0=Idle, 1=Running, 2=Fault

    Notes: Includes optional low/high PV “hold” with hysteresis (normal-stop class).
*)

FUNCTION_BLOCK FB_WirePitControl
VAR_INPUT
    // ===== Sequence commands =====
    startCommand                 : BOOL;            // Start pulse toggles RUN latch
    stopCommand                  : BOOL;            // Stop pulse/level forces stop

    // ===== Manual output & Auto SP nudge =====
    processSetpointManInc        : BOOL;            // Manual output ↑ (0..100%)
    processSetpointManDec        : BOOL;            // Manual output ↓ (0..100%)
    processSetpointManSteps      : REAL := 0.1;

    processSetpointAutoInc       : BOOL;            // Auto SP ↑ (engineering units or %)
    processSetpointAutoDec       : BOOL;            // Auto SP ↓ (engineering units or %)
    processSetpointAutoSteps     : REAL := 1.0;

    // ===== Mode =====
    autoMode                     : BOOL;            // TRUE=Automatic / FALSE=Manual
    reverseActing                : BOOL := FALSE;   // TRUE: higher output decreases PV; FALSE: direct

    // ===== Process signals (PV in engineering units) =====
    wirePitLevel           : REAL;            // PV (engineering units), e.g., bar/kPa/°C/…
	whiteWaterSiloLevel			: REAL;
    // ===== PID parameters (OSCAT CTRL_PID) =====
    kp                           : REAL := 1.0;     // Proportional gain (sign handled via reverseActing)
    tn                           : REAL := 8.0;     // Integral time [s]
    tv                           : REAL := 0.0;     // Derivative time [s]

    // ===== Output limits & offset =====
    outLowLimitPct               : REAL := 0.0;     // Min output %
    outHighLimitPct              : REAL := 100.0;   // Max output %
    outputOffsetPct              : REAL := 0.0;     // Offset added to final output

    // ===== PID housekeeping =====
    resetPID                     : BOOL;            // Reset integrator

    // ===== Input filter (OSCAT FT_PT1) =====
    enableInputFilter            : BOOL := TRUE;    // Enable PV PT1 filter
    inputFilterTime              : TIME := T#300ms; // PT1 time constant
    inputFilterGainK             : REAL := 1.0;     // PT1 gain

    displayFilterTime            : TIME := T#20ms;  // Small PT1 for HMI displays

    // ===== Optional scaling (engineering ↔ %) =====
    enableScaling                : BOOL := TRUE;    // Enable engineering↔% scaling
    pLoEng                       : REAL := 0.0;     // Engineering low bound
    pHiEng                       : REAL := 10.0;    // Engineering high bound

